KUKA KRL program: EPS_2_26115_SA6999_A_20260219035531.src

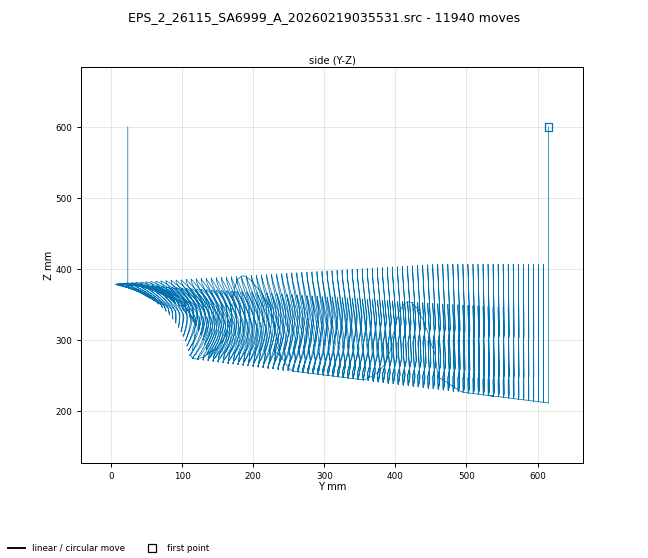
[picture p0: tool path of EPS_2_26115_SA6999_A_20260219035531.src, 11940 of 11942 moves have a stored position in this frame; points joined in program order, loops and branches not executed]
&ACCESS RVP
&REL 4
&COMMENT QRS 19112012
&PARAM EDITMASK = *
DEF PART()
EXT BAS (BAS_COMMAND :IN,REAL :IN )
INT I
BAS (#INITMOV,0 )

;KUKA QRS Post kuka4.cps  Date:22-06-2017 !

File_ID=3054

QRS_PRE_INIT()

;Init var - Until changes are made in qrs_pre_init
Outlet_Square_prg=0
Inlet_1_Square_prg=0
Inlet_2_Square_prg=0
Inlet_3_Square_prg=0
Inlet_4_Square_prg=0
Inlet_5_Square_prg=0

Outlet_1={X 0.000, Y 460.000, Z 306.500, B 0.000, E1 0.000 }
Inlet_1={X 0.000, Y 536.220, Z 246.500, B 0.000, E1 184.000 }
Outlet_1_type=201
Inlet_1_type=201
;QRS#1=Sidecore dimensions
;QRS#2=200-8" PVC SDR 35 Cut Back
;QRS#3=200-8" PVC SDR 35
;QRS#4=
;QRS#5=
;QRS#6=
;QRS#7=
;QRS#8=
;QRS#9=12-08 PSX
;QRS#10=12-08 PSX
;QRS#11=
;QRS#12=
;QRS#13=
;QRS#14=
;QRS#15=
;QRS#16=1220x127x686 2,25'
;QRS#17=EPS Height
;QRS#18=407
;QRS#19=*
;QRS#20= UPDATED VERSION 22-06-2017
;QRS#21=*
Outlet_Square=0100
Inlet_1_Square=0100
Inlet_2_Square=0
Inlet_3_Square=0
Inlet_4_Square=0
Inlet_5_Square=0
Mill_Square=1
Outlet_Square_Prg=214
Inlet_1_Square_prg=204

QRS_INIT()

$ADVANCE=5

; T1
PTP {E1 173.66,E2 173.66}
PTP {X 0,Y 615.427,A -85,B 0,C 180,E1 173.66,E2 173.66,E3 0,E4 0,E5 0,E6 0}
QRS_SPEED_INIT()
LIN {X 0,Y 615.427,Z 600,A -85,B 0,C 180,E1 173.66,E2 173.66,E3 0,E4 0,E5 0,E6 0} C_VEL
LIN {X 0,Y 615.427,Z 221.878,A -85,B 0,C 180,E1 173.66,E2 173.66} C_VEL
LIN {X 0,Y 615.427,Z 213.7,A -85,B 0,C 180,E1 173.66,E2 173.66} C_VEL
LIN {X 0,Y 615.43,Z 211.7,A -85,B 0,C 180,E1 173.474,E2 173.474} C_VEL
LIN {X 0,Y 615.497,Z 211.695,A -85,B 0,C 180,E1 170.801,E2 170.801} C_VEL
LIN {X 0,Y 615.455,Z 211.694,A -85,B 0,C 180,E1 168.138,E2 168.138} C_VEL
LIN {X 0,Y 615.489,Z 211.696,A -85,B 0,C 180,E1 165.451,E2 165.451} C_VEL
LIN {X 0,Y 615.486,Z 211.688,A -85,B 0,C 180,E1 162.729,E2 162.729} C_VEL
LIN {X 0,Y 615.47,Z 211.696,A -85,B 0,C 180,E1 159.966,E2 159.966} C_VEL
LIN {X 0,Y 615.456,Z 211.693,A -85,B 0,C 180,E1 157.663,E2 157.663} C_VEL
LIN {X 0,Y 615.492,Z 211.702,A -85,B 0,C 180,E1 155.008,E2 155.008} C_VEL
LIN {X 0,Y 615.434,Z 211.7,A -85,B 0,C 180,E1 152.082,E2 152.082} C_VEL
LIN {X 0,Y 615.48,Z 211.7,A -85,B 0,C 180,E1 149.839,E2 149.839} C_VEL
LIN {X 0,Y 615.492,Z 211.691,A -85,B 0,C 180,E1 147.543,E2 147.543} C_VEL
LIN {X 0,Y 615.479,Z 211.688,A -85,B 0,C 180,E1 145.184,E2 145.184} C_VEL
LIN {X 0,Y 615.487,Z 211.698,A -85,B 0,C 180,E1 142.757,E2 142.757} C_VEL
LIN {X 0,Y 615.474,Z 211.689,A -85,B 0,C 180,E1 139.914,E2 139.914} C_VEL
LIN {X 0,Y 615.464,Z 211.698,A -85,B 0,C 180,E1 136.956,E2 136.956} C_VEL
LIN {X 0,Y 615.438,Z 211.7,A -85,B 0,C 180,E1 134.926,E2 134.926} C_VEL
LIN {X 0,Y 615.479,Z 211.7,A -85,B 0,C 180,E1 132.079,E2 132.079} C_VEL
LIN {X 0,Y 615.481,Z 211.692,A -85,B 0,C 180,E1 129.752,E2 129.752} C_VEL
LIN {X 0,Y 615.472,Z 211.697,A -85,B 0,C 180,E1 126.934,E2 126.934} C_VEL
LIN {X 0,Y 615.495,Z 211.685,A -85,B 0,C 180,E1 124.022,E2 124.022} C_VEL
LIN {X 0,Y 615.482,Z 211.693,A -85,B 0,C 180,E1 121.687,E2 121.687} C_VEL
LIN {X 0,Y 615.499,Z 213.244,A -85,B 0,C 180,E1 120.16,E2 120.16} C_VEL
LIN {X 0,Y 615.488,Z 215.951,A -85,B 0,C 180,E1 117.916,E2 117.916} C_VEL
LIN {X 0,Y 615.438,Z 218.768,A -85,B 0,C 180,E1 115.558,E2 115.558} C_VEL
LIN {X 0,Y 615.427,Z 221.262,A -85,B 0,C 180,E1 113.56,E2 113.56} C_VEL
LIN {X 0,Y 615.431,Z 224.037,A -85,B 0,C 180,E1 111.435,E2 111.435} C_VEL
LIN {X 0,Y 615.492,Z 227.738,A -85,B 0,C 180,E1 108.647,E2 108.647} C_VEL
LIN {X 0,Y 615.445,Z 231.467,A -85,B 0,C 180,E1 105.907,E2 105.907} C_VEL
LIN {X 0,Y 615.482,Z 235.206,A -85,B 0,C 180,E1 103.202,E2 103.202} C_VEL
LIN {X 0,Y 615.478,Z 238.945,A -85,B 0,C 180,E1 100.528,E2 100.528} C_VEL
LIN {X 0,Y 615.461,Z 242.721,A -85,B 0,C 180,E1 97.877,E2 97.877} C_VEL
LIN {X 0,Y 615.484,Z 243.188,A -85,B 0,C 180,E1 97.546,E2 97.546} C_VEL
LIN {X 0,Y 615.492,Z 257.399,A -85,B 0,C 180,E1 97.217,E2 97.217} C_VEL
LIN {X 0,Y 615.498,Z 269.488,A -85,B 0,C 180,E1 96.809,E2 96.809} C_VEL
LIN {X 0,Y 615.463,Z 280.578,A -85,B 0,C 180,E1 96.311,E2 96.311} C_VEL
LIN {X 0,Y 615.485,Z 291.97,A -85,B 0,C 180,E1 95.653,E2 95.653} C_VEL
LIN {X 0,Y 615.498,Z 302.233,A -85,B 0,C 180,E1 94.914,E2 94.914} C_VEL
LIN {X 0,Y 615.499,Z 311.516,A -85,B 0,C 180,E1 94.093,E2 94.093} C_VEL
LIN {X 0,Y 615.498,Z 320.461,A -85,B 0,C 180,E1 93.11,E2 93.11} C_VEL
LIN {X 0,Y 615.497,Z 327.686,A -85,B 0,C 180,E1 92.128,E2 92.128} C_VEL
LIN {X 0,Y 615.497,Z 334.314,A -85,B 0,C 180,E1 90.982,E2 90.982} C_VEL
LIN {X 0,Y 615.495,Z 338.703,A -85,B 0,C 180,E1 90.001,E2 90.001} C_VEL
LIN {X 0,Y 615.496,Z 341.018,A -85,B 0,C 180,E1 89.347,E2 89.347} C_VEL
LIN {X 0,Y 615.495,Z 342.915,A -85,B 0,C 180,E1 88.692,E2 88.692} C_VEL
LIN {X 0,Y 615.5,Z 344.4,A -85,B 0,C 180,E1 88.038,E2 88.038} C_VEL
LIN {X 0,Y 615.496,Z 346.089,A -85,B 0,C 180,E1 86.728,E2 86.728} C_VEL
LIN {X 0,Y 615.496,Z 346.254,A -85,B 0,C 180,E1 85.417,E2 85.417} C_VEL
LIN {X 0,Y 615.496,Z 344.792,A -85,B 0,C 180,E1 84.103,E2 84.103} C_VEL
LIN {X 0,Y 615.496,Z 343.421,A -85,B 0,C 180,E1 83.418,E2 83.418} C_VEL
LIN {X 0,Y 615.496,Z 340.674,A -85,B 0,C 180,E1 82.456,E2 82.456} C_VEL
LIN {X 0,Y 615.497,Z 336.845,A -85,B 0,C 180,E1 81.465,E2 81.465} C_VEL
LIN {X 0,Y 615.496,Z 331.874,A -85,B 0,C 180,E1 80.471,E2 80.471} C_VEL
LIN {X 0,Y 615.497,Z 325.603,A -85,B 0,C 180,E1 79.474,E2 79.474} C_VEL
LIN {X 0,Y 615.496,Z 317.715,A -85,B 0,C 180,E1 78.474,E2 78.474} C_VEL
LIN {X 0,Y 615.498,Z 309.63,A -85,B 0,C 180,E1 77.639,E2 77.639} C_VEL
LIN {X 0,Y 615.499,Z 299.733,A -85,B 0,C 180,E1 76.8,E2 76.8} C_VEL
LIN {X 0,Y 615.476,Z 289.065,A -85,B 0,C 180,E1 76.073,E2 76.073} C_VEL
LIN {X 0,Y 615.488,Z 277.524,A -85,B 0,C 180,E1 75.452,E2 75.452} C_VEL
LIN {X 0,Y 615.481,Z 265.299,A -85,B 0,C 180,E1 74.944,E2 74.944} C_VEL
LIN {X 0,Y 615.492,Z 252.488,A -85,B 0,C 180,E1 74.563,E2 74.563} C_VEL
LIN {X 0,Y 615.484,Z 243.199,A -85,B 0,C 180,E1 74.372,E2 74.372} C_VEL
LIN {X 0,Y 615.472,Z 239.89,A -85,B 0,C 180,E1 72.044,E2 72.044} C_VEL
LIN {X 0,Y 615.488,Z 235.979,A -85,B 0,C 180,E1 69.27,E2 69.27} C_VEL
LIN {X 0,Y 615.464,Z 232.076,A -85,B 0,C 180,E1 66.444,E2 66.444} C_VEL
LIN {X 0,Y 615.461,Z 229.123,A -85,B 0,C 180,E1 64.284,E2 64.284} C_VEL
LIN {X 0,Y 615.491,Z 225.444,A -85,B 0,C 180,E1 61.55,E2 61.55} C_VEL
LIN {X 0,Y 615.457,Z 222.002,A -85,B 0,C 180,E1 58.919,E2 58.919} C_VEL
LIN {X 0,Y 615.45,Z 218.911,A -85,B 0,C 180,E1 56.472,E2 56.472} C_VEL
LIN {X 0,Y 615.45,Z 215.467,A -85,B 0,C 180,E1 53.574,E2 53.574} C_VEL
LIN {X 0,Y 615.464,Z 212.279,A -85,B 0,C 180,E1 50.941,E2 50.941} C_VEL
LIN {X 0,Y 615.482,Z 211.69,A -85,B 0,C 180,E1 49.912,E2 49.912} C_VEL
LIN {X 0,Y 615.483,Z 211.694,A -85,B 0,C 180,E1 47.648,E2 47.648} C_VEL
LIN {X 0,Y 615.456,Z 211.696,A -85,B 0,C 180,E1 44.93,E2 44.93} C_VEL
LIN {X 0,Y 615.465,Z 211.7,A -85,B 0,C 180,E1 42.08,E2 42.08} C_VEL
LIN {X 0,Y 615.46,Z 211.695,A -85,B 0,C 180,E1 39.753,E2 39.753} C_VEL
LIN {X 0,Y 615.48,Z 211.693,A -85,B 0,C 180,E1 36.938,E2 36.938} C_VEL
LIN {X 0,Y 615.488,Z 211.7,A -85,B 0,C 180,E1 34.022,E2 34.022} C_VEL
LIN {X 0,Y 615.437,Z 211.7,A -85,B 0,C 180,E1 31.689,E2 31.689} C_VEL
LIN {X 0,Y 615.471,Z 211.7,A -85,B 0,C 180,E1 29.407,E2 29.407} C_VEL
LIN {X 0,Y 615.484,Z 211.691,A -85,B 0,C 180,E1 26.445,E2 26.445} C_VEL
LIN {X 0,Y 615.477,Z 211.699,A -85,B 0,C 180,E1 24.009,E2 24.009} C_VEL
LIN {X 0,Y 615.446,Z 211.7,A -85,B 0,C 180,E1 21.434,E2 21.434} C_VEL
LIN {X 0,Y 615.467,Z 211.694,A -85,B 0,C 180,E1 18.603,E2 18.603} C_VEL
LIN {X 0,Y 615.487,Z 211.7,A -85,B 0,C 180,E1 15.905,E2 15.905} C_VEL
LIN {X 0,Y 615.49,Z 211.69,A -85,B 0,C 180,E1 13.201,E2 13.201} C_VEL
LIN {X 0,Y 615.443,Z 211.701,A -85,B 0,C 180,E1 10.528,E2 10.528} C_VEL
LIN {X 0,Y 615.479,Z 211.701,A -85,B 0,C 180,E1 7.876,E2 7.876} C_VEL
LIN {X 0,Y 615.492,Z 211.688,A -85,B 0,C 180,E1 5.241,E2 5.241} C_VEL
LIN {X 0,Y 615.477,Z 211.699,A -85,B 0,C 180,E1 2.618,E2 2.618} C_VEL
LIN {X 0,Y 615.448,Z 211.7,A -85,B 0,C 180,E1 0,E2 0} C_VEL
LIN {X 0,Y 615.48,Z 211.693,A -85,B 0,C 180,E1 -2.618,E2 -2.618} C_VEL
LIN {X 0,Y 615.486,Z 211.698,A -85,B 0,C 180,E1 -5.241,E2 -5.241} C_VEL
LIN {X 0,Y 615.467,Z 211.693,A -85,B 0,C 180,E1 -7.876,E2 -7.876} C_VEL
LIN {X 0,Y 615.478,Z 211.7,A -85,B 0,C 180,E1 -10.527,E2 -10.527} C_VEL
LIN {X 0,Y 615.456,Z 211.699,A -85,B 0,C 180,E1 -13.202,E2 -13.202} C_VEL
LIN {X 0,Y 615.492,Z 211.689,A -85,B 0,C 180,E1 -15.905,E2 -15.905} C_VEL
LIN {X 0,Y 615.489,Z 211.701,A -85,B 0,C 180,E1 -18.646,E2 -18.646} C_VEL
LIN {X 0,Y 615.448,Z 211.7,A -85,B 0,C 180,E1 -20.732,E2 -20.732} C_VEL
LIN {X 0,Y 615.485,Z 211.703,A -85,B 0,C 180,E1 -23.556,E2 -23.556} C_VEL
LIN {X 0,Y 615.476,Z 211.695,A -85,B 0,C 180,E1 -26.445,E2 -26.445} C_VEL
LIN {X 0,Y 615.48,Z 211.699,A -85,B 0,C 180,E1 -28.658,E2 -28.658} C_VEL
LIN {X 0,Y 615.452,Z 211.697,A -85,B 0,C 180,E1 -31.083,E2 -31.083} C_VEL
LIN {X 0,Y 615.456,Z 211.697,A -85,B 0,C 180,E1 -34.024,E2 -34.024} C_VEL
LIN {X 0,Y 615.475,Z 211.697,A -85,B 0,C 180,E1 -36.426,E2 -36.426} C_VEL
LIN {X 0,Y 615.478,Z 211.691,A -85,B 0,C 180,E1 -39.063,E2 -39.063} C_VEL
LIN {X 0,Y 615.497,Z 211.695,A -85,B 0,C 180,E1 -41.473,E2 -41.473} C_VEL
LIN {X 0,Y 615.436,Z 211.7,A -85,B 0,C 180,E1 -44.154,E2 -44.154} C_VEL
LIN {X 0,Y 615.493,Z 211.697,A -85,B 0,C 180,E1 -46.758,E2 -46.758} C_VEL
LIN {X 0,Y 615.483,Z 211.692,A -85,B 0,C 180,E1 -49.395,E2 -49.395} C_VEL
LIN {X 0,Y 615.457,Z 211.698,A -85,B 0,C 180,E1 -51.992,E2 -51.992} C_VEL
LIN {X 0,Y 615.462,Z 211.822,A -85,B 0,C 180,E1 -54.535,E2 -54.535} C_VEL
LIN {X 0,Y 615.471,Z 220.583,A -85,B 0,C 180,E1 -57.154,E2 -57.154} C_VEL
LIN {X 0,Y 615.452,Z 228.516,A -85,B 0,C 180,E1 -59.46,E2 -59.46} C_VEL
LIN {X 0,Y 615.483,Z 237.76,A -85,B 0,C 180,E1 -62.086,E2 -62.086} C_VEL
LIN {X 0,Y 615.488,Z 247.269,A -85,B 0,C 180,E1 -64.721,E2 -64.721} C_VEL
LIN {X 0,Y 615.475,Z 256.241,A -85,B 0,C 180,E1 -67.156,E2 -67.156} C_VEL
LIN {X 0,Y 615.489,Z 264.799,A -85,B 0,C 180,E1 -69.443,E2 -69.443} C_VEL
LIN {X 0,Y 615.49,Z 276.018,A -85,B 0,C 180,E1 -72.388,E2 -72.388} C_VEL
LIN {X 0,Y 615.479,Z 286.546,A -85,B 0,C 180,E1 -75.114,E2 -75.114} C_VEL
LIN {X 0,Y 615.444,Z 295.77,A -85,B 0,C 180,E1 -77.47,E2 -77.47} C_VEL
LIN {X 0,Y 615.499,Z 299.212,A -85,B 0,C 180,E1 -78.349,E2 -78.349} C_VEL
LIN {X 0,Y 615.497,Z 313.861,A -85,B 0,C 180,E1 -78.641,E2 -78.641} C_VEL
LIN {X 0,Y 615.451,Z 327.004,A -85,B 0,C 180,E1 -79.052,E2 -79.052} C_VEL
LIN {X 0,Y 615.438,Z 338.796,A -85,B 0,C 180,E1 -79.556,E2 -79.556} C_VEL
LIN {X 0,Y 615.482,Z 349.407,A -85,B 0,C 180,E1 -80.139,E2 -80.139} C_VEL
LIN {X 0,Y 615.498,Z 360.245,A -85,B 0,C 180,E1 -80.885,E2 -80.885} C_VEL
LIN {X 0,Y 615.497,Z 370.823,A -85,B 0,C 180,E1 -81.795,E2 -81.795} C_VEL
LIN {X 0,Y 615.497,Z 379.974,A -85,B 0,C 180,E1 -82.785,E2 -82.785} C_VEL
LIN {X 0,Y 615.497,Z 387.322,A -85,B 0,C 180,E1 -83.774,E2 -83.774} C_VEL
LIN {X 0,Y 615.498,Z 393.21,A -85,B 0,C 180,E1 -84.76,E2 -84.76} C_VEL
LIN {X 0,Y 615.493,Z 397.856,A -85,B 0,C 180,E1 -85.745,E2 -85.745} C_VEL
LIN {X 0,Y 615.494,Z 401.402,A -85,B 0,C 180,E1 -86.728,E2 -86.728} C_VEL
LIN {X 0,Y 615.497,Z 403.235,A -85,B 0,C 180,E1 -87.383,E2 -87.383} C_VEL
LIN {X 0,Y 615.5,Z 404.609,A -85,B 0,C 180,E1 -88.038,E2 -88.038} C_VEL
LIN {X 0,Y 615.496,Z 406.174,A -85,B 0,C 180,E1 -89.347,E2 -89.347} C_VEL
LIN {X 0,Y 615.494,Z 406.389,A -85,B 0,C 180,E1 -90.001,E2 -90.001} C_VEL
LIN {X 0,Y 615.495,Z 405.579,A -85,B 0,C 180,E1 -91.31,E2 -91.31} C_VEL
LIN {X 0,Y 615.5,Z 404.606,A -85,B 0,C 180,E1 -91.964,E2 -91.964} C_VEL
LIN {X 0,Y 615.497,Z 403.231,A -85,B 0,C 180,E1 -92.619,E2 -92.619} C_VEL
LIN {X 0,Y 615.496,Z 400.346,A -85,B 0,C 180,E1 -93.602,E2 -93.602} C_VEL
LIN {X 0,Y 615.498,Z 396.437,A -85,B 0,C 180,E1 -94.585,E2 -94.585} C_VEL
LIN {X 0,Y 615.499,Z 391.4,A -85,B 0,C 180,E1 -95.571,E2 -95.571} C_VEL
LIN {X 0,Y 615.497,Z 384.869,A -85,B 0,C 180,E1 -96.583,E2 -96.583} C_VEL
LIN {X 0,Y 615.497,Z 377.125,A -85,B 0,C 180,E1 -97.546,E2 -97.546} C_VEL
LIN {X 0,Y 615.498,Z 369.035,A -85,B 0,C 180,E1 -98.372,E2 -98.372} C_VEL
LIN {X 0,Y 615.499,Z 359.155,A -85,B 0,C 180,E1 -99.2,E2 -99.2} C_VEL
LIN {X 0,Y 615.471,Z 347.969,A -85,B 0,C 180,E1 -99.946,E2 -99.946} C_VEL
LIN {X 0,Y 615.437,Z 337.012,A -85,B 0,C 180,E1 -100.529,E2 -100.529} C_VEL
LIN {X 0,Y 615.457,Z 324.782,A -85,B 0,C 180,E1 -101.03,E2 -101.03} C_VEL
LIN {X 0,Y 615.499,Z 312.023,A -85,B 0,C 180,E1 -101.402,E2 -101.402} C_VEL
LIN {X 0,Y 615.498,Z 299.205,A -85,B 0,C 180,E1 -101.653,E2 -101.653} C_VEL
LIN {X 0,Y 615.454,Z 289.085,A -85,B 0,C 180,E1 -104.238,E2 -104.238} C_VEL
LIN {X 0,Y 615.491,Z 278.636,A -85,B 0,C 180,E1 -106.929,E2 -106.929} C_VEL
LIN {X 0,Y 615.482,Z 268.101,A -85,B 0,C 180,E1 -109.686,E2 -109.686} C_VEL
LIN {X 0,Y 615.49,Z 258.087,A -85,B 0,C 180,E1 -112.346,E2 -112.346} C_VEL
LIN {X 0,Y 615.477,Z 248.318,A -85,B 0,C 180,E1 -114.993,E2 -114.993} C_VEL
LIN {X 0,Y 615.492,Z 239.071,A -85,B 0,C 180,E1 -117.546,E2 -117.546} C_VEL
LIN {X 0,Y 615.456,Z 229.83,A -85,B 0,C 180,E1 -120.163,E2 -120.163} C_VEL
LIN {X 0,Y 615.445,Z 221.899,A -85,B 0,C 180,E1 -122.461,E2 -122.461} C_VEL
LIN {X 0,Y 615.491,Z 212.64,A -85,B 0,C 180,E1 -125.215,E2 -125.215} C_VEL
LIN {X 0,Y 615.453,Z 211.7,A -85,B 0,C 180,E1 -125.519,E2 -125.519} C_VEL
LIN {X 0,Y 615.435,Z 211.699,A -85,B 0,C 180,E1 -128.073,E2 -128.073} C_VEL
LIN {X 0,Y 615.495,Z 211.697,A -85,B 0,C 180,E1 -130.607,E2 -130.607} C_VEL
LIN {X 0,Y 615.467,Z 211.691,A -85,B 0,C 180,E1 -133.247,E2 -133.247} C_VEL
LIN {X 0,Y 615.487,Z 211.696,A -85,B 0,C 180,E1 -136.004,E2 -136.004} C_VEL
LIN {X 0,Y 615.489,Z 211.69,A -85,B 0,C 180,E1 -138.906,E2 -138.906} C_VEL
LIN {X 0,Y 615.493,Z 211.701,A -85,B 0,C 180,E1 -141.096,E2 -141.096} C_VEL
LIN {X 0,Y 615.443,Z 211.697,A -85,B 0,C 180,E1 -143.572,E2 -143.572} C_VEL
LIN {X 0,Y 615.492,Z 211.701,A -85,B 0,C 180,E1 -146.466,E2 -146.466} C_VEL
LIN {X 0,Y 615.441,Z 211.697,A -85,B 0,C 180,E1 -149.078,E2 -149.078} C_VEL
LIN {X 0,Y 615.474,Z 211.699,A -85,B 0,C 180,E1 -151.553,E2 -151.553} C_VEL
LIN {X 0,Y 615.482,Z 211.687,A -85,B 0,C 180,E1 -154.434,E2 -154.434} C_VEL
LIN {X 0,Y 615.485,Z 211.701,A -85,B 0,C 180,E1 -157.155,E2 -157.155} C_VEL
LIN {X 0,Y 615.484,Z 211.688,A -85,B 0,C 180,E1 -159.967,E2 -159.967} C_VEL
LIN {X 0,Y 615.461,Z 211.699,A -85,B 0,C 180,E1 -162.729,E2 -162.729} C_VEL
LIN {X 0,Y 615.439,Z 211.699,A -85,B 0,C 180,E1 -164.773,E2 -164.773} C_VEL
LIN {X 0,Y 615.427,Z 211.7,A -85,B 0,C 180,E1 -166.797,E2 -166.797} C_VEL
LIN {X 0,Y 615.489,Z 211.701,A -85,B 0,C 180,E1 -169.473,E2 -169.473} C_VEL
LIN {X 0,Y 615.466,Z 211.691,A -85,B 0,C 180,E1 -172.124,E2 -172.124} C_VEL
LIN {X 0,Y 615.488,Z 211.7,A -85,B 0,C 180,E1 -174.759,E2 -174.759} C_VEL
LIN {X 0,Y 615.487,Z 211.687,A -85,B 0,C 180,E1 -177.382,E2 -177.382} C_VEL
LIN {X 0,Y 615.493,Z 211.697,A -85,B 0,C 180,E1 -180,E2 -180} C_VEL
LIN {X 0,Y 615.449,Z 211.696,A -85,B 0,C 180,E1 -182.618,E2 -182.618} C_VEL
LIN {X 0,Y 615.485,Z 211.696,A -85,B 0,C 180,E1 -185.241,E2 -185.241} C_VEL
LIN {X 0,Y 615.43,Z 211.7,A -85,B 0,C 180,E1 -186.526,E2 -186.526} C_VEL
LIN {X 0,Y 614.797,Z 211.849,A -85,B 0,C 180,E1 -187.072,E2 -187.072} C_VEL
LIN {X 0,Y 612.005,Z 212.247,A -85,B 0,C 180,E1 -187.958,E2 -187.958} C_VEL
LIN {X 0,Y 609.615,Z 212.56,A -85,B 0,C 180,E1 -188.671,E2 -188.671} C_VEL
LIN {X 0,Y 608.56,Z 212.682,A -85,B 0,C 180,E1 -189.22,E2 -189.22} C_VEL
LIN {X 0,Y 608.46,Z 212.691,A -85,B 0,C 180,E1 -189.406,E2 -189.406} C_VEL
LIN {X 0,Y 608.442,Z 212.692,A -85,B 0,C 180,E1 -192,E2 -192} C_VEL
LIN {X 0,Y 608.479,Z 212.689,A -85,B 0,C 180,E1 -194.721,E2 -194.721} C_VEL
LIN {X 0,Y 608.455,Z 212.692,A -85,B 0,C 180,E1 -197.477,E2 -197.477} C_VEL
LIN {X 0,Y 608.448,Z 212.691,A -85,B 0,C 180,E1 -200.275,E2 -200.275} C_VEL
LIN {X 0,Y 608.436,Z 212.692,A -85,B 0,C 180,E1 -202.469,E2 -202.469} C_VEL
LIN {X 0,Y 608.425,Z 212.697,A -85,B 0,C 180,E1 -205.302,E2 -205.302} C_VEL
LIN {X 0,Y 608.432,Z 212.696,A -85,B 0,C 180,E1 -208.268,E2 -208.268} C_VEL
LIN {X 0,Y 608.443,Z 212.695,A -85,B 0,C 180,E1 -210.547,E2 -210.547} C_VEL
LIN {X 0,Y 608.45,Z 212.69,A -85,B 0,C 180,E1 -212.88,E2 -212.88} C_VEL
LIN {X 0,Y 608.447,Z 212.693,A -85,B 0,C 180,E1 -215.278,E2 -215.278} C_VEL
LIN {X 0,Y 608.465,Z 212.691,A -85,B 0,C 180,E1 -217.747,E2 -217.747} C_VEL
LIN {X 0,Y 608.448,Z 212.691,A -85,B 0,C 180,E1 -220.328,E2 -220.328} C_VEL
LIN {X 0,Y 608.435,Z 212.697,A -85,B 0,C 180,E1 -222.962,E2 -222.962} C_VEL
LIN {X 0,Y 608.424,Z 212.694,A -85,B 0,C 180,E1 -225.74,E2 -225.74} C_VEL
LIN {X 0,Y 608.427,Z 212.693,A -85,B 0,C 180,E1 -228.662,E2 -228.662} C_VEL
LIN {X 0,Y 608.424,Z 212.699,A -85,B 0,C 180,E1 -231.408,E2 -231.408} C_VEL
LIN {X 0,Y 608.453,Z 212.691,A -85,B 0,C 180,E1 -233.954,E2 -233.954} C_VEL
LIN {X 0,Y 608.45,Z 212.691,A -85,B 0,C 180,E1 -236.328,E2 -236.328} C_VEL
LIN {X 0,Y 608.42,Z 212.777,A -85,B 0,C 180,E1 -238.737,E2 -238.737} C_VEL
LIN {X 0,Y 608.427,Z 215.467,A -85,B 0,C 180,E1 -240.977,E2 -240.977} C_VEL
LIN {X 0,Y 608.423,Z 219.032,A -85,B 0,C 180,E1 -243.963,E2 -243.963} C_VEL
LIN {X 0,Y 608.395,Z 221.656,A -85,B 0,C 180,E1 -246.151,E2 -246.151} C_VEL
LIN {X 0,Y 608.373,Z 224.447,A -85,B 0,C 180,E1 -248.304,E2 -248.304} C_VEL
LIN {X 0,Y 608.374,Z 227.247,A -85,B 0,C 180,E1 -250.426,E2 -250.426} C_VEL
LIN {X 0,Y 608.412,Z 230.992,A -85,B 0,C 180,E1 -253.214,E2 -253.214} C_VEL
LIN {X 0,Y 608.385,Z 234.831,A -85,B 0,C 180,E1 -256.017,E2 -256.017} C_VEL
LIN {X 0,Y 608.419,Z 238.526,A -85,B 0,C 180,E1 -258.674,E2 -258.674} C_VEL
LIN {X 0,Y 608.409,Z 242.313,A -85,B 0,C 180,E1 -261.362,E2 -261.362} C_VEL
LIN {X 0,Y 608.422,Z 243.754,A -85,B 0,C 180,E1 -262.334,E2 -262.334} C_VEL
LIN {X 0,Y 608.527,Z 256.976,A -85,B 0,C 180,E1 -262.638,E2 -262.638} C_VEL
LIN {X 0,Y 608.527,Z 269.893,A -85,B 0,C 180,E1 -263.076,E2 -263.076} C_VEL
LIN {X 0,Y 608.476,Z 282.377,A -85,B 0,C 180,E1 -263.657,E2 -263.657} C_VEL
LIN {X 0,Y 608.498,Z 294.157,A -85,B 0,C 180,E1 -264.365,E2 -264.365} C_VEL
LIN {X 0,Y 608.476,Z 303.085,A -85,B 0,C 180,E1 -265.03,E2 -265.03} C_VEL
LIN {X 0,Y 608.474,Z 312.286,A -85,B 0,C 180,E1 -265.859,E2 -265.859} C_VEL
LIN {X 0,Y 608.459,Z 321.215,A -85,B 0,C 180,E1 -266.854,E2 -266.854} C_VEL
LIN {X 0,Y 608.454,Z 328.428,A -85,B 0,C 180,E1 -267.848,E2 -267.848} C_VEL
LIN {X 0,Y 608.449,Z 333.311,A -85,B 0,C 180,E1 -268.675,E2 -268.675} C_VEL
LIN {X 0,Y 608.442,Z 338.067,A -85,B 0,C 180,E1 -269.668,E2 -269.668} C_VEL
LIN {X 0,Y 608.439,Z 341.722,A -85,B 0,C 180,E1 -270.661,E2 -270.661} C_VEL
LIN {X 0,Y 608.448,Z 343.613,A -85,B 0,C 180,E1 -271.323,E2 -271.323} C_VEL
LIN {X 0,Y 608.444,Z 345.077,A -85,B 0,C 180,E1 -271.985,E2 -271.985} C_VEL
LIN {X 0,Y 608.422,Z 346.732,A -85,B 0,C 180,E1 -273.31,E2 -273.31} C_VEL
LIN {X 0,Y 608.433,Z 346.989,A -85,B 0,C 180,E1 -273.973,E2 -273.973} C_VEL
LIN {X 0,Y 608.429,Z 346.833,A -85,B 0,C 180,E1 -274.637,E2 -274.637} C_VEL
LIN {X 0,Y 608.433,Z 345.309,A -85,B 0,C 180,E1 -275.966,E2 -275.966} C_VEL
LIN {X 0,Y 608.447,Z 343.956,A -85,B 0,C 180,E1 -276.632,E2 -276.632} C_VEL
LIN {X 0,Y 608.427,Z 341.073,A -85,B 0,C 180,E1 -277.633,E2 -277.633} C_VEL
LIN {X 0,Y 608.431,Z 337.153,A -85,B 0,C 180,E1 -278.635,E2 -278.635} C_VEL
LIN {X 0,Y 608.435,Z 332.078,A -85,B 0,C 180,E1 -279.641,E2 -279.641} C_VEL
LIN {X 0,Y 608.443,Z 325.68,A -85,B 0,C 180,E1 -280.649,E2 -280.649} C_VEL
LIN {X 0,Y 608.474,Z 317.634,A -85,B 0,C 180,E1 -281.66,E2 -281.66} C_VEL
LIN {X 0,Y 608.468,Z 309.411,A -85,B 0,C 180,E1 -282.506,E2 -282.506} C_VEL
LIN {X 0,Y 608.482,Z 299.346,A -85,B 0,C 180,E1 -283.355,E2 -283.355} C_VEL
LIN {X 0,Y 608.479,Z 287.907,A -85,B 0,C 180,E1 -284.121,E2 -284.121} C_VEL
LIN {X 0,Y 608.51,Z 276.663,A -85,B 0,C 180,E1 -284.719,E2 -284.719} C_VEL
LIN {X 0,Y 608.516,Z 264.051,A -85,B 0,C 180,E1 -285.232,E2 -285.232} C_VEL
LIN {X 0,Y 608.552,Z 251.421,A -85,B 0,C 180,E1 -285.596,E2 -285.596} C_VEL
LIN {X 0,Y 608.429,Z 243.67,A -85,B 0,C 180,E1 -285.771,E2 -285.771} C_VEL
LIN {X 0,Y 608.426,Z 239.526,A -85,B 0,C 180,E1 -288.702,E2 -288.702} C_VEL
LIN {X 0,Y 608.416,Z 236.341,A -85,B 0,C 180,E1 -290.982,E2 -290.982} C_VEL
LIN {X 0,Y 608.418,Z 233.383,A -85,B 0,C 180,E1 -293.124,E2 -293.124} C_VEL
LIN {X 0,Y 608.408,Z 229.424,A -85,B 0,C 180,E1 -296.036,E2 -296.036} C_VEL
LIN {X 0,Y 608.426,Z 225.448,A -85,B 0,C 180,E1 -299.021,E2 -299.021} C_VEL
LIN {X 0,Y 608.401,Z 222.454,A -85,B 0,C 180,E1 -301.319,E2 -301.319} C_VEL
LIN {X 0,Y 608.42,Z 219.508,A -85,B 0,C 180,E1 -303.727,E2 -303.727} C_VEL
LIN {X 0,Y 608.436,Z 216.719,A -85,B 0,C 180,E1 -306.091,E2 -306.091} C_VEL
LIN {X 0,Y 608.417,Z 213.704,A -85,B 0,C 180,E1 -308.59,E2 -308.59} C_VEL
LIN {X 0,Y 608.41,Z 212.703,A -85,B 0,C 180,E1 -309.443,E2 -309.443} C_VEL
LIN {X 0,Y 608.465,Z 212.689,A -85,B 0,C 180,E1 -312.059,E2 -312.059} C_VEL
LIN {X 0,Y 608.432,Z 212.695,A -85,B 0,C 180,E1 -314.796,E2 -314.796} C_VEL
LIN {X 0,Y 608.412,Z 212.696,A -85,B 0,C 180,E1 -317.036,E2 -317.036} C_VEL
LIN {X 0,Y 608.445,Z 212.694,A -85,B 0,C 180,E1 -319.696,E2 -319.696} C_VEL
LIN {X 0,Y 608.463,Z 212.692,A -85,B 0,C 180,E1 -322.253,E2 -322.253} C_VEL
LIN {X 0,Y 608.468,Z 212.689,A -85,B 0,C 180,E1 -325.09,E2 -325.09} C_VEL
LIN {X 0,Y 608.448,Z 212.694,A -85,B 0,C 180,E1 -327.904,E2 -327.904} C_VEL
LIN {X 0,Y 608.435,Z 212.693,A -85,B 0,C 180,E1 -330.218,E2 -330.218} C_VEL
LIN {X 0,Y 608.477,Z 212.691,A -85,B 0,C 180,E1 -332.79,E2 -332.79} C_VEL
LIN {X 0,Y 608.453,Z 212.693,A -85,B 0,C 180,E1 -335.429,E2 -335.429} C_VEL
LIN {X 0,Y 608.431,Z 212.693,A -85,B 0,C 180,E1 -338.307,E2 -338.307} C_VEL
LIN {X 0,Y 608.456,Z 212.691,A -85,B 0,C 180,E1 -341.284,E2 -341.284} C_VEL
LIN {X 0,Y 608.457,Z 212.696,A -85,B 0,C 180,E1 -343.906,E2 -343.906} C_VEL
LIN {X 0,Y 608.462,Z 212.69,A -85,B 0,C 180,E1 -346.643,E2 -346.643} C_VEL
LIN {X 0,Y 608.434,Z 212.695,A -85,B 0,C 180,E1 -349.349,E2 -349.349} C_VEL
LIN {X 0,Y 608.466,Z 212.693,A -85,B 0,C 180,E1 -352.033,E2 -352.033} C_VEL
LIN {X 0,Y 608.47,Z 212.688,A -85,B 0,C 180,E1 -354.698,E2 -354.698} C_VEL
LIN {X 0,Y 608.469,Z 212.694,A -85,B 0,C 180,E1 -357.352,E2 -357.352} C_VEL
LIN {X 0,Y 608.441,Z 212.693,A -85,B 0,C 180,E1 -360,E2 -360} C_VEL
LIN {X 0,Y 608.47,Z 212.69,A -85,B 0,C 180,E1 -362.648,E2 -362.648} C_VEL
LIN {X 0,Y 608.464,Z 212.695,A -85,B 0,C 180,E1 -365.302,E2 -365.302} C_VEL
LIN {X 0,Y 608.463,Z 212.689,A -85,B 0,C 180,E1 -367.967,E2 -367.967} C_VEL
LIN {X 0,Y 608.445,Z 212.695,A -85,B 0,C 180,E1 -370.65,E2 -370.65} C_VEL
LIN {X 0,Y 608.443,Z 212.695,A -85,B 0,C 180,E1 -373.357,E2 -373.357} C_VEL
LIN {X 0,Y 608.461,Z 212.69,A -85,B 0,C 180,E1 -376.094,E2 -376.094} C_VEL
LIN {X 0,Y 608.447,Z 212.695,A -85,B 0,C 180,E1 -378.87,E2 -378.87} C_VEL
LIN {X 0,Y 608.441,Z 212.697,A -85,B 0,C 180,E1 -381.693,E2 -381.693} C_VEL
LIN {X 0,Y 608.438,Z 212.693,A -85,B 0,C 180,E1 -384.572,E2 -384.572} C_VEL
LIN {X 0,Y 608.475,Z 212.69,A -85,B 0,C 180,E1 -387.209,E2 -387.209} C_VEL
LIN {X 0,Y 608.475,Z 212.693,A -85,B 0,C 180,E1 -389.975,E2 -389.975} C_VEL
LIN {X 0,Y 608.433,Z 212.694,A -85,B 0,C 180,E1 -392.881,E2 -392.881} C_VEL
LIN {X 0,Y 608.437,Z 212.697,A -85,B 0,C 180,E1 -395.278,E2 -395.278} C_VEL
LIN {X 0,Y 608.466,Z 212.689,A -85,B 0,C 180,E1 -397.747,E2 -397.747} C_VEL
LIN {X 0,Y 608.441,Z 212.695,A -85,B 0,C 180,E1 -400.33,E2 -400.33} C_VEL
LIN {X 0,Y 608.476,Z 212.696,A -85,B 0,C 180,E1 -403.311,E2 -403.311} C_VEL
LIN {X 0,Y 608.448,Z 212.693,A -85,B 0,C 180,E1 -406.13,E2 -406.13} C_VEL
LIN {X 0,Y 608.455,Z 212.691,A -85,B 0,C 180,E1 -408.825,E2 -408.825} C_VEL
LIN {X 0,Y 608.466,Z 212.695,A -85,B 0,C 180,E1 -411.413,E2 -411.413} C_VEL
LIN {X 0,Y 608.426,Z 212.695,A -85,B 0,C 180,E1 -413.957,E2 -413.957} C_VEL
LIN {X 0,Y 608.448,Z 212.82,A -85,B 0,C 180,E1 -414.369,E2 -414.369} C_VEL
LIN {X 0,Y 608.514,Z 221.921,A -85,B 0,C 180,E1 -417.125,E2 -417.125} C_VEL
LIN {X 0,Y 608.499,Z 229.865,A -85,B 0,C 180,E1 -419.458,E2 -419.458} C_VEL
LIN {X 0,Y 608.495,Z 239.132,A -85,B 0,C 180,E1 -422.112,E2 -422.112} C_VEL
LIN {X 0,Y 608.479,Z 248.399,A -85,B 0,C 180,E1 -424.702,E2 -424.702} C_VEL
LIN {X 0,Y 608.476,Z 258.99,A -85,B 0,C 180,E1 -427.596,E2 -427.596} C_VEL
LIN {X 0,Y 608.457,Z 269.581,A -85,B 0,C 180,E1 -430.431,E2 -430.431} C_VEL
LIN {X 0,Y 608.449,Z 280.173,A -85,B 0,C 180,E1 -433.217,E2 -433.217} C_VEL
LIN {X 0,Y 608.435,Z 290.896,A -85,B 0,C 180,E1 -435.997,E2 -435.997} C_VEL
LIN {X 0,Y 608.437,Z 299.576,A -85,B 0,C 180,E1 -438.223,E2 -438.223} C_VEL
LIN {X 0,Y 608.549,Z 313.14,A -85,B 0,C 180,E1 -438.489,E2 -438.489} C_VEL
LIN {X 0,Y 608.485,Z 325.548,A -85,B 0,C 180,E1 -438.866,E2 -438.866} C_VEL
LIN {X 0,Y 608.444,Z 337.194,A -85,B 0,C 180,E1 -439.351,E2 -439.351} C_VEL
LIN {X 0,Y 608.471,Z 349.596,A -85,B 0,C 180,E1 -440.024,E2 -440.024} C_VEL
LIN {X 0,Y 608.483,Z 360.487,A -85,B 0,C 180,E1 -440.779,E2 -440.779} C_VEL
LIN {X 0,Y 608.474,Z 371.123,A -85,B 0,C 180,E1 -441.7,E2 -441.7} C_VEL
LIN {X 0,Y 608.47,Z 378.969,A -85,B 0,C 180,E1 -442.535,E2 -442.535} C_VEL
LIN {X 0,Y 608.46,Z 386.29,A -85,B 0,C 180,E1 -443.485,E2 -443.485} C_VEL
LIN {X 0,Y 608.45,Z 391.871,A -85,B 0,C 180,E1 -444.367,E2 -444.367} C_VEL
LIN {X 0,Y 608.432,Z 396.954,A -85,B 0,C 180,E1 -445.363,E2 -445.363} C_VEL
LIN {X 0,Y 608.449,Z 400.899,A -85,B 0,C 180,E1 -446.359,E2 -446.359} C_VEL
LIN {X 0,Y 608.425,Z 403.812,A -85,B 0,C 180,E1 -447.353,E2 -447.353} C_VEL
LIN {X 0,Y 608.444,Z 405.203,A -85,B 0,C 180,E1 -448.015,E2 -448.015} C_VEL
LIN {X 0,Y 608.438,Z 406.784,A -85,B 0,C 180,E1 -449.339,E2 -449.339} C_VEL
LIN {X 0,Y 608.434,Z 407,A -85,B 0,C 180,E1 -450.001,E2 -450.001} C_VEL
LIN {X 0,Y 608.448,Z 406.183,A -85,B 0,C 180,E1 -451.325,E2 -451.325} C_VEL
LIN {X 0,Y 608.445,Z 405.2,A -85,B 0,C 180,E1 -451.987,E2 -451.987} C_VEL
LIN {X 0,Y 608.425,Z 403.807,A -85,B 0,C 180,E1 -452.649,E2 -452.649} C_VEL
LIN {X 0,Y 608.449,Z 400.893,A -85,B 0,C 180,E1 -453.643,E2 -453.643} C_VEL
LIN {X 0,Y 608.432,Z 396.946,A -85,B 0,C 180,E1 -454.639,E2 -454.639} C_VEL
LIN {X 0,Y 608.438,Z 390.871,A -85,B 0,C 180,E1 -455.802,E2 -455.802} C_VEL
LIN {X 0,Y 608.463,Z 384.228,A -85,B 0,C 180,E1 -456.8,E2 -456.8} C_VEL
LIN {X 0,Y 608.456,Z 375.981,A -85,B 0,C 180,E1 -457.801,E2 -457.801} C_VEL
LIN {X 0,Y 608.472,Z 367.525,A -85,B 0,C 180,E1 -458.637,E2 -458.637} C_VEL
LIN {X 0,Y 608.48,Z 357.078,A -85,B 0,C 180,E1 -459.474,E2 -459.474} C_VEL
LIN {X 0,Y 608.482,Z 346.74,A -85,B 0,C 180,E1 -460.146,E2 -460.146} C_VEL
LIN {X 0,Y 608.463,Z 335.863,A -85,B 0,C 180,E1 -460.713,E2 -460.713} C_VEL
LIN {X 0,Y 608.492,Z 324.079,A -85,B 0,C 180,E1 -461.187,E2 -461.187} C_VEL
LIN {X 0,Y 608.551,Z 311.227,A -85,B 0,C 180,E1 -461.555,E2 -461.555} C_VEL
LIN {X 0,Y 608.439,Z 299.527,A -85,B 0,C 180,E1 -461.79,E2 -461.79} C_VEL
LIN {X 0,Y 608.405,Z 289.432,A -85,B 0,C 180,E1 -464.381,E2 -464.381} C_VEL
LIN {X 0,Y 608.451,Z 280.165,A -85,B 0,C 180,E1 -466.785,E2 -466.785} C_VEL
LIN {X 0,Y 608.458,Z 269.574,A -85,B 0,C 180,E1 -469.571,E2 -469.571} C_VEL
LIN {X 0,Y 608.465,Z 258.722,A -85,B 0,C 180,E1 -472.477,E2 -472.477} C_VEL
LIN {X 0,Y 608.479,Z 248.391,A -85,B 0,C 180,E1 -475.301,E2 -475.301} C_VEL
LIN {X 0,Y 608.496,Z 239.124,A -85,B 0,C 180,E1 -477.89,E2 -477.89} C_VEL
LIN {X 0,Y 608.481,Z 229.857,A -85,B 0,C 180,E1 -480.545,E2 -480.545} C_VEL
LIN {X 0,Y 608.528,Z 220.59,A -85,B 0,C 180,E1 -483.271,E2 -483.271} C_VEL
LIN {X 0,Y 608.426,Z 212.697,A -85,B 0,C 180,E1 -485.673,E2 -485.673} C_VEL
LIN {X 0,Y 608.434,Z 212.694,A -85,B 0,C 180,E1 -488.236,E2 -488.236} C_VEL
LIN {X 0,Y 608.44,Z 212.691,A -85,B 0,C 180,E1 -491.179,E2 -491.179} C_VEL
LIN {X 0,Y 608.469,Z 212.694,A -85,B 0,C 180,E1 -493.87,E2 -493.87} C_VEL
LIN {X 0,Y 608.483,Z 212.686,A -85,B 0,C 180,E1 -496.691,E2 -496.691} C_VEL
LIN {X 0,Y 608.459,Z 212.692,A -85,B 0,C 180,E1 -499.697,E2 -499.697} C_VEL
LIN {X 0,Y 608.481,Z 212.694,A -85,B 0,C 180,E1 -502.841,E2 -502.841} C_VEL
LIN {X 0,Y 608.426,Z 212.693,A -85,B 0,C 180,E1 -505.528,E2 -505.528} C_VEL
LIN {X 0,Y 608.439,Z 212.695,A -85,B 0,C 180,E1 -507.904,E2 -507.904} C_VEL
LIN {X 0,Y 608.481,Z 212.691,A -85,B 0,C 180,E1 -510.221,E2 -510.221} C_VEL
LIN {X 0,Y 608.438,Z 212.695,A -85,B 0,C 180,E1 -513.225,E2 -513.225} C_VEL
LIN {X 0,Y 608.478,Z 212.688,A -85,B 0,C 180,E1 -515.849,E2 -515.849} C_VEL
LIN {X 0,Y 608.468,Z 212.689,A -85,B 0,C 180,E1 -518.308,E2 -518.308} C_VEL
LIN {X 0,Y 608.447,Z 212.692,A -85,B 0,C 180,E1 -521.13,E2 -521.13} C_VEL
LIN {X 0,Y 608.454,Z 212.694,A -85,B 0,C 180,E1 -523.906,E2 -523.906} C_VEL
LIN {X 0,Y 608.42,Z 212.694,A -85,B 0,C 180,E1 -526.643,E2 -526.643} C_VEL
LIN {X 0,Y 608.454,Z 212.695,A -85,B 0,C 180,E1 -529.35,E2 -529.35} C_VEL
LIN {X 0,Y 608.437,Z 212.692,A -85,B 0,C 180,E1 -532.033,E2 -532.033} C_VEL
LIN {X 0,Y 608.467,Z 212.694,A -85,B 0,C 180,E1 -534.698,E2 -534.698} C_VEL
LIN {X 0,Y 608.478,Z 212.686,A -85,B 0,C 180,E1 -537.352,E2 -537.352} C_VEL
LIN {X 0,Y 608.484,Z 212.692,A -85,B 0,C 180,E1 -540,E2 -540} C_VEL
LIN {X 0,Y 608.445,Z 212.691,A -85,B 0,C 180,E1 -542.648,E2 -542.648} C_VEL
LIN {X 0,Y 608.461,Z 212.694,A -85,B 0,C 180,E1 -545.302,E2 -545.302} C_VEL
LIN {X 0,Y 608.406,Z 212.695,A -85,B 0,C 180,E1 -547.968,E2 -547.968} C_VEL
LIN {X 0,Y 608.46,Z 212.691,A -85,B 0,C 180,E1 -549.406,E2 -549.406} C_VEL
LIN {X 0,Y 607.755,Z 212.778,A -85,B 0,C 180,E1 -549.959,E2 -549.959} C_VEL
LIN {X 0,Y 604.894,Z 213.141,A -85,B 0,C 180,E1 -550.856,E2 -550.856} C_VEL
LIN {X 0,Y 602.504,Z 213.436,A -85,B 0,C 180,E1 -551.577,E2 -551.577} C_VEL
LIN {X 0,Y 601.484,Z 213.56,A -85,B 0,C 180,E1 -552.134,E2 -552.134} C_VEL
LIN {X 0,Y 601.403,Z 213.57,A -85,B 0,C 180,E1 -552.322,E2 -552.322} C_VEL
LIN {X 0,Y 601.434,Z 213.565,A -85,B 0,C 180,E1 -554.897,E2 -554.897} C_VEL
LIN {X 0,Y 601.419,Z 213.566,A -85,B 0,C 180,E1 -556.986,E2 -556.986} C_VEL
LIN {X 0,Y 601.401,Z 213.574,A -85,B 0,C 180,E1 -559.81,E2 -559.81} C_VEL
LIN {X 0,Y 601.408,Z 213.569,A -85,B 0,C 180,E1 -562.683,E2 -562.683} C_VEL
LIN {X 0,Y 601.386,Z 213.577,A -85,B 0,C 180,E1 -564.88,E2 -564.88} C_VEL
LIN {X 0,Y 601.377,Z 213.572,A -85,B 0,C 180,E1 -567.354,E2 -567.354} C_VEL
LIN {X 0,Y 601.384,Z 213.57,A -85,B 0,C 180,E1 -569.395,E2 -569.395} C_VEL
LIN {X 0,Y 601.401,Z 213.571,A -85,B 0,C 180,E1 -571.727,E2 -571.727} C_VEL
LIN {X 0,Y 601.426,Z 213.569,A -85,B 0,C 180,E1 -574.119,E2 -574.119} C_VEL
LIN {X 0,Y 601.404,Z 213.568,A -85,B 0,C 180,E1 -576.583,E2 -576.583} C_VEL
LIN {X 0,Y 601.41,Z 213.575,A -85,B 0,C 180,E1 -579.127,E2 -579.127} C_VEL
LIN {X 0,Y 601.417,Z 213.566,A -85,B 0,C 180,E1 -581.766,E2 -581.766} C_VEL
LIN {X 0,Y 601.405,Z 213.576,A -85,B 0,C 180,E1 -584.532,E2 -584.532} C_VEL
LIN {X 0,Y 601.357,Z 213.574,A -85,B 0,C 180,E1 -587.324,E2 -587.324} C_VEL
LIN {X 0,Y 601.404,Z 213.573,A -85,B 0,C 180,E1 -590.003,E2 -590.003} C_VEL
LIN {X 0,Y 601.436,Z 213.564,A -85,B 0,C 180,E1 -592.618,E2 -592.618} C_VEL
LIN {X 0,Y 601.418,Z 213.573,A -85,B 0,C 180,E1 -595.067,E2 -595.067} C_VEL
LIN {X 0,Y 601.427,Z 213.566,A -85,B 0,C 180,E1 -597.483,E2 -597.483} C_VEL
LIN {X 0,Y 601.345,Z 213.809,A -85,B 0,C 180,E1 -599.053,E2 -599.053} C_VEL
LIN {X 0,Y 601.358,Z 216.577,A -85,B 0,C 180,E1 -601.368,E2 -601.368} C_VEL
LIN {X 0,Y 601.344,Z 219.852,A -85,B 0,C 180,E1 -604.147,E2 -604.147} C_VEL
LIN {X 0,Y 601.304,Z 222.744,A -85,B 0,C 180,E1 -606.584,E2 -606.584} C_VEL
LIN {X 0,Y 601.343,Z 226.385,A -85,B 0,C 180,E1 -609.474,E2 -609.474} C_VEL
LIN {X 0,Y 601.311,Z 229.19,A -85,B 0,C 180,E1 -611.604,E2 -611.604} C_VEL
LIN {X 0,Y 601.33,Z 232.002,A -85,B 0,C 180,E1 -613.709,E2 -613.709} C_VEL
LIN {X 0,Y 601.311,Z 235.765,A -85,B 0,C 180,E1 -616.481,E2 -616.481} C_VEL
LIN {X 0,Y 601.333,Z 239.541,A -85,B 0,C 180,E1 -619.221,E2 -619.221} C_VEL
LIN {X 0,Y 601.318,Z 243.568,A -85,B 0,C 180,E1 -622.106,E2 -622.106} C_VEL
LIN {X 0,Y 601.308,Z 243.687,A -85,B 0,C 180,E1 -622.19,E2 -622.19} C_VEL
LIN {X 0,Y 601.606,Z 247.938,A -85,B 0,C 180,E1 -622.278,E2 -622.278} C_VEL
LIN {X 0,Y 601.568,Z 260.67,A -85,B 0,C 180,E1 -622.616,E2 -622.616} C_VEL
LIN {X 0,Y 601.551,Z 273.95,A -85,B 0,C 180,E1 -623.121,E2 -623.121} C_VEL
LIN {X 0,Y 601.48,Z 285.059,A -85,B 0,C 180,E1 -623.68,E2 -623.68} C_VEL
LIN {X 0,Y 601.468,Z 296.038,A -85,B 0,C 180,E1 -624.383,E2 -624.383} C_VEL
LIN {X 0,Y 601.44,Z 305.612,A -85,B 0,C 180,E1 -625.139,E2 -625.139} C_VEL
LIN {X 0,Y 601.401,Z 314.362,A -85,B 0,C 180,E1 -625.978,E2 -625.978} C_VEL
LIN {X 0,Y 601.384,Z 322.91,A -85,B 0,C 180,E1 -626.985,E2 -626.985} C_VEL
LIN {X 0,Y 601.355,Z 329.761,A -85,B 0,C 180,E1 -627.99,E2 -627.99} C_VEL
LIN {X 0,Y 601.382,Z 335.259,A -85,B 0,C 180,E1 -628.995,E2 -628.995} C_VEL
LIN {X 0,Y 601.357,Z 339.584,A -85,B 0,C 180,E1 -629.999,E2 -629.999} C_VEL
LIN {X 0,Y 601.341,Z 341.873,A -85,B 0,C 180,E1 -630.669,E2 -630.669} C_VEL
LIN {X 0,Y 601.348,Z 343.74,A -85,B 0,C 180,E1 -631.338,E2 -631.338} C_VEL
LIN {X 0,Y 601.343,Z 345.156,A -85,B 0,C 180,E1 -632.008,E2 -632.008} C_VEL
LIN {X 0,Y 601.338,Z 346.766,A -85,B 0,C 180,E1 -633.349,E2 -633.349} C_VEL
LIN {X 0,Y 601.342,Z 346.999,A -85,B 0,C 180,E1 -634.02,E2 -634.02} C_VEL
LIN {X 0,Y 601.336,Z 346.208,A -85,B 0,C 180,E1 -635.364,E2 -635.364} C_VEL
LIN {X 0,Y 601.362,Z 344.103,A -85,B 0,C 180,E1 -636.594,E2 -636.594} C_VEL
LIN {X 0,Y 601.339,Z 340.92,A -85,B 0,C 180,E1 -637.723,E2 -637.723} C_VEL
LIN {X 0,Y 601.35,Z 336.949,A -85,B 0,C 180,E1 -638.738,E2 -638.738} C_VEL
LIN {X 0,Y 601.361,Z 330.812,A -85,B 0,C 180,E1 -639.925,E2 -639.925} C_VEL
LIN {X 0,Y 601.386,Z 323.751,A -85,B 0,C 180,E1 -640.991,E2 -640.991} C_VEL
LIN {X 0,Y 601.43,Z 315.698,A -85,B 0,C 180,E1 -641.97,E2 -641.97} C_VEL
LIN {X 0,Y 601.426,Z 307.032,A -85,B 0,C 180,E1 -642.827,E2 -642.827} C_VEL
LIN {X 0,Y 601.476,Z 296.842,A -85,B 0,C 180,E1 -643.648,E2 -643.648} C_VEL
LIN {X 0,Y 601.503,Z 285.652,A -85,B 0,C 180,E1 -644.375,E2 -644.375} C_VEL
LIN {X 0,Y 601.528,Z 273.702,A -85,B 0,C 180,E1 -644.98,E2 -644.98} C_VEL
LIN {X 0,Y 601.54,Z 261.232,A -85,B 0,C 180,E1 -645.457,E2 -645.457} C_VEL
LIN {X 0,Y 601.599,Z 248.366,A -85,B 0,C 180,E1 -645.802,E2 -645.802} C_VEL
LIN {X 0,Y 601.328,Z 243.711,A -85,B 0,C 180,E1 -645.897,E2 -645.897} C_VEL
LIN {X 0,Y 601.342,Z 239.64,A -85,B 0,C 180,E1 -648.796,E2 -648.796} C_VEL
LIN {X 0,Y 601.311,Z 236.268,A -85,B 0,C 180,E1 -651.242,E2 -651.242} C_VEL
LIN {X 0,Y 601.332,Z 233.309,A -85,B 0,C 180,E1 -653.413,E2 -653.413} C_VEL
LIN {X 0,Y 601.312,Z 230.04,A -85,B 0,C 180,E1 -655.847,E2 -655.847} C_VEL
LIN {X 0,Y 601.343,Z 226.366,A -85,B 0,C 180,E1 -658.63,E2 -658.63} C_VEL
LIN {X 0,Y 601.334,Z 222.781,A -85,B 0,C 180,E1 -661.441,E2 -661.441} C_VEL
LIN {X 0,Y 601.353,Z 219.686,A -85,B 0,C 180,E1 -664.122,E2 -664.122} C_VEL
LIN {X 0,Y 601.333,Z 216.757,A -85,B 0,C 180,E1 -666.586,E2 -666.586} C_VEL
LIN {X 0,Y 601.37,Z 213.729,A -85,B 0,C 180,E1 -669.128,E2 -669.128} C_VEL
LIN {X 0,Y 601.424,Z 213.566,A -85,B 0,C 180,E1 -671.764,E2 -671.764} C_VEL
LIN {X 0,Y 601.419,Z 213.572,A -85,B 0,C 180,E1 -674.534,E2 -674.534} C_VEL
LIN {X 0,Y 601.405,Z 213.573,A -85,B 0,C 180,E1 -677.408,E2 -677.408} C_VEL
LIN {X 0,Y 601.406,Z 213.57,A -85,B 0,C 180,E1 -680.466,E2 -680.466} C_VEL
LIN {X 0,Y 601.43,Z 213.573,A -85,B 0,C 180,E1 -682.617,E2 -682.617} C_VEL
LIN {X 0,Y 601.426,Z 213.566,A -85,B 0,C 180,E1 -685.068,E2 -685.068} C_VEL
LIN {X 0,Y 601.431,Z 213.572,A -85,B 0,C 180,E1 -687.484,E2 -687.484} C_VEL
LIN {X 0,Y 601.4,Z 213.573,A -85,B 0,C 180,E1 -690.606,E2 -690.606} C_VEL
LIN {X 0,Y 601.449,Z 213.565,A -85,B 0,C 180,E1 -692.889,E2 -692.889} C_VEL
LIN {X 0,Y 601.451,Z 213.569,A -85,B 0,C 180,E1 -695.859,E2 -695.859} C_VEL
LIN {X 0,Y 601.384,Z 213.574,A -85,B 0,C 180,E1 -698.76,E2 -698.76} C_VEL
LIN {X 0,Y 601.388,Z 213.571,A -85,B 0,C 180,E1 -701.607,E2 -701.607} C_VEL
LIN {X 0,Y 601.433,Z 213.568,A -85,B 0,C 180,E1 -703.713,E2 -703.713} C_VEL
LIN {X 0,Y 601.413,Z 213.568,A -85,B 0,C 180,E1 -706.484,E2 -706.484} C_VEL
LIN {X 0,Y 601.404,Z 213.572,A -85,B 0,C 180,E1 -709.224,E2 -709.224} C_VEL
LIN {X 0,Y 601.427,Z 213.569,A -85,B 0,C 180,E1 -711.939,E2 -711.939} C_VEL
LIN {X 0,Y 601.434,Z 213.565,A -85,B 0,C 180,E1 -714.636,E2 -714.636} C_VEL
LIN {X 0,Y 601.434,Z 213.57,A -85,B 0,C 180,E1 -717.321,E2 -717.321} C_VEL
LIN {X 0,Y 601.412,Z 213.569,A -85,B 0,C 180,E1 -720,E2 -720} C_VEL
LIN {X 0,Y 601.434,Z 213.566,A -85,B 0,C 180,E1 -722.679,E2 -722.679} C_VEL
LIN {X 0,Y 601.426,Z 213.573,A -85,B 0,C 180,E1 -725.364,E2 -725.364} C_VEL
LIN {X 0,Y 601.428,Z 213.566,A -85,B 0,C 180,E1 -728.061,E2 -728.061} C_VEL
LIN {X 0,Y 601.39,Z 213.571,A -85,B 0,C 180,E1 -731.002,E2 -731.002} C_VEL
LIN {X 0,Y 601.401,Z 213.574,A -85,B 0,C 180,E1 -733.516,E2 -733.516} C_VEL
LIN {X 0,Y 601.435,Z 213.565,A -85,B 0,C 180,E1 -736.287,E2 -736.287} C_VEL
LIN {X 0,Y 601.407,Z 213.569,A -85,B 0,C 180,E1 -739.099,E2 -739.099} C_VEL
LIN {X 0,Y 601.38,Z 213.572,A -85,B 0,C 180,E1 -741.24,E2 -741.24} C_VEL
LIN {X 0,Y 601.445,Z 213.564,A -85,B 0,C 180,E1 -744.141,E2 -744.141} C_VEL
LIN {X 0,Y 601.447,Z 213.567,A -85,B 0,C 180,E1 -747.111,E2 -747.111} C_VEL
LIN {X 0,Y 601.42,Z 213.567,A -85,B 0,C 180,E1 -749.393,E2 -749.393} C_VEL
LIN {X 0,Y 601.385,Z 213.578,A -85,B 0,C 180,E1 -751.728,E2 -751.728} C_VEL
LIN {X 0,Y 601.415,Z 213.568,A -85,B 0,C 180,E1 -754.119,E2 -754.119} C_VEL
LIN {X 0,Y 601.399,Z 213.575,A -85,B 0,C 180,E1 -756.583,E2 -756.583} C_VEL
LIN {X 0,Y 601.435,Z 213.566,A -85,B 0,C 180,E1 -759.537,E2 -759.537} C_VEL
LIN {X 0,Y 601.408,Z 213.574,A -85,B 0,C 180,E1 -761.767,E2 -761.767} C_VEL
LIN {X 0,Y 601.389,Z 213.572,A -85,B 0,C 180,E1 -764.533,E2 -764.533} C_VEL
LIN {X 0,Y 601.406,Z 213.569,A -85,B 0,C 180,E1 -767.41,E2 -767.41} C_VEL
LIN {X 0,Y 601.41,Z 213.574,A -85,B 0,C 180,E1 -770.006,E2 -770.006} C_VEL
LIN {X 0,Y 601.428,Z 213.567,A -85,B 0,C 180,E1 -772.619,E2 -772.619} C_VEL
LIN {X 0,Y 601.402,Z 213.692,A -85,B 0,C 180,E1 -774.159,E2 -774.159} C_VEL
LIN {X 0,Y 601.541,Z 219.274,A -85,B 0,C 180,E1 -775.89,E2 -775.89} C_VEL
LIN {X 0,Y 601.561,Z 228.025,A -85,B 0,C 180,E1 -778.524,E2 -778.524} C_VEL
LIN {X 0,Y 601.478,Z 237.808,A -85,B 0,C 180,E1 -781.377,E2 -781.377} C_VEL
LIN {X 0,Y 601.477,Z 247.454,A -85,B 0,C 180,E1 -784.121,E2 -784.121} C_VEL
LIN {X 0,Y 601.465,Z 256.342,A -85,B 0,C 180,E1 -786.593,E2 -786.593} C_VEL
LIN {X 0,Y 601.43,Z 266.934,A -85,B 0,C 180,E1 -789.479,E2 -789.479} C_VEL
LIN {X 0,Y 601.4,Z 277.525,A -85,B 0,C 180,E1 -792.313,E2 -792.313} C_VEL
LIN {X 0,Y 601.365,Z 288.116,A -85,B 0,C 180,E1 -795.103,E2 -795.103} C_VEL
LIN {X 0,Y 601.338,Z 297.383,A -85,B 0,C 180,E1 -797.514,E2 -797.514} C_VEL
LIN {X 0,Y 601.372,Z 299.534,A -85,B 0,C 180,E1 -798.072,E2 -798.072} C_VEL
LIN {X 0,Y 601.592,Z 313.14,A -85,B 0,C 180,E1 -798.354,E2 -798.354} C_VEL
LIN {X 0,Y 601.509,Z 326.352,A -85,B 0,C 180,E1 -798.766,E2 -798.766} C_VEL
LIN {X 0,Y 601.468,Z 338.944,A -85,B 0,C 180,E1 -799.311,E2 -799.311} C_VEL
LIN {X 0,Y 601.461,Z 349.597,A -85,B 0,C 180,E1 -799.907,E2 -799.907} C_VEL
LIN {X 0,Y 601.449,Z 360.488,A -85,B 0,C 180,E1 -800.67,E2 -800.67} C_VEL
LIN {X 0,Y 601.429,Z 371.123,A -85,B 0,C 180,E1 -801.602,E2 -801.602} C_VEL
LIN {X 0,Y 601.417,Z 378.969,A -85,B 0,C 180,E1 -802.447,E2 -802.447} C_VEL
LIN {X 0,Y 601.369,Z 386.23,A -85,B 0,C 180,E1 -803.399,E2 -803.399} C_VEL
LIN {X 0,Y 601.372,Z 391.872,A -85,B 0,C 180,E1 -804.3,E2 -804.3} C_VEL
LIN {X 0,Y 601.336,Z 396.954,A -85,B 0,C 180,E1 -805.308,E2 -805.308} C_VEL
LIN {X 0,Y 601.368,Z 400.899,A -85,B 0,C 180,E1 -806.316,E2 -806.316} C_VEL
LIN {X 0,Y 601.325,Z 403.812,A -85,B 0,C 180,E1 -807.321,E2 -807.321} C_VEL
LIN {X 0,Y 601.343,Z 405.203,A -85,B 0,C 180,E1 -807.992,E2 -807.992} C_VEL
LIN {X 0,Y 601.339,Z 406.784,A -85,B 0,C 180,E1 -809.331,E2 -809.331} C_VEL
LIN {X 0,Y 601.335,Z 407,A -85,B 0,C 180,E1 -810.001,E2 -810.001} C_VEL
LIN {X 0,Y 601.347,Z 406.183,A -85,B 0,C 180,E1 -811.34,E2 -811.34} C_VEL
LIN {X 0,Y 601.343,Z 405.2,A -85,B 0,C 180,E1 -812.01,E2 -812.01} C_VEL
LIN {X 0,Y 601.325,Z 403.807,A -85,B 0,C 180,E1 -812.681,E2 -812.681} C_VEL
LIN {X 0,Y 601.368,Z 400.893,A -85,B 0,C 180,E1 -813.686,E2 -813.686} C_VEL
LIN {X 0,Y 601.336,Z 396.946,A -85,B 0,C 180,E1 -814.694,E2 -814.694} C_VEL
LIN {X 0,Y 601.373,Z 390.871,A -85,B 0,C 180,E1 -815.87,E2 -815.87} C_VEL
LIN {X 0,Y 601.382,Z 384.228,A -85,B 0,C 180,E1 -816.881,E2 -816.881} C_VEL
LIN {X 0,Y 601.401,Z 375.981,A -85,B 0,C 180,E1 -817.893,E2 -817.893} C_VEL
LIN {X 0,Y 601.436,Z 367.526,A -85,B 0,C 180,E1 -818.739,E2 -818.739} C_VEL
LIN {X 0,Y 601.447,Z 357.078,A -85,B 0,C 180,E1 -819.586,E2 -819.586} C_VEL
LIN {X 0,Y 601.473,Z 346.74,A -85,B 0,C 180,E1 -820.265,E2 -820.265} C_VEL
LIN {X 0,Y 601.482,Z 335.241,A -85,B 0,C 180,E1 -820.868,E2 -820.868} C_VEL
LIN {X 0,Y 601.528,Z 322.313,A -85,B 0,C 180,E1 -821.376,E2 -821.376} C_VEL
LIN {X 0,Y 601.597,Z 309.399,A -85,B 0,C 180,E1 -821.733,E2 -821.733} C_VEL
LIN {X 0,Y 601.373,Z 299.527,A -85,B 0,C 180,E1 -821.93,E2 -821.93} C_VEL
LIN {X 0,Y 601.37,Z 289.432,A -85,B 0,C 180,E1 -824.553,E2 -824.553} C_VEL
LIN {X 0,Y 601.396,Z 278.841,A -85,B 0,C 180,E1 -827.338,E2 -827.338} C_VEL
LIN {X 0,Y 601.421,Z 268.25,A -85,B 0,C 180,E1 -830.166,E2 -830.166} C_VEL
LIN {X 0,Y 601.436,Z 258.983,A -85,B 0,C 180,E1 -832.683,E2 -832.683} C_VEL
LIN {X 0,Y 601.463,Z 249.715,A -85,B 0,C 180,E1 -835.246,E2 -835.246} C_VEL
LIN {X 0,Y 601.504,Z 240.448,A -85,B 0,C 180,E1 -837.864,E2 -837.864} C_VEL
LIN {X 0,Y 601.507,Z 231.181,A -85,B 0,C 180,E1 -840.548,E2 -840.548} C_VEL
LIN {X 0,Y 601.585,Z 221.914,A -85,B 0,C 180,E1 -843.305,E2 -843.305} C_VEL
LIN {X 0,Y 601.585,Z 215.919,A -85,B 0,C 180,E1 -845.137,E2 -845.137} C_VEL
LIN {X 0,Y 601.388,Z 213.574,A -85,B 0,C 180,E1 -845.933,E2 -845.933} C_VEL
LIN {X 0,Y 601.4,Z 213.574,A -85,B 0,C 180,E1 -848.467,E2 -848.467} C_VEL
LIN {X 0,Y 601.405,Z 213.57,A -85,B 0,C 180,E1 -850.876,E2 -850.876} C_VEL
LIN {X 0,Y 601.412,Z 213.569,A -85,B 0,C 180,E1 -853.589,E2 -853.589} C_VEL
LIN {X 0,Y 601.436,Z 213.564,A -85,B 0,C 180,E1 -856.428,E2 -856.428} C_VEL
LIN {X 0,Y 601.415,Z 213.571,A -85,B 0,C 180,E1 -859.125,E2 -859.125} C_VEL
LIN {X 0,Y 601.4,Z 213.569,A -85,B 0,C 180,E1 -861.73,E2 -861.73} C_VEL
LIN {X 0,Y 601.38,Z 213.573,A -85,B 0,C 180,E1 -864.245,E2 -864.245} C_VEL
LIN {X 0,Y 601.407,Z 213.572,A -85,B 0,C 180,E1 -866.685,E2 -866.685} C_VEL
LIN {X 0,Y 601.394,Z 213.569,A -85,B 0,C 180,E1 -869.056,E2 -869.056} C_VEL
LIN {X 0,Y 601.415,Z 213.569,A -85,B 0,C 180,E1 -871.372,E2 -871.372} C_VEL
LIN {X 0,Y 601.419,Z 213.566,A -85,B 0,C 180,E1 -874.382,E2 -874.382} C_VEL
LIN {X 0,Y 601.399,Z 213.57,A -85,B 0,C 180,E1 -876.589,E2 -876.589} C_VEL
LIN {X 0,Y 601.421,Z 213.566,A -85,B 0,C 180,E1 -879.478,E2 -879.478} C_VEL
LIN {X 0,Y 601.388,Z 213.577,A -85,B 0,C 180,E1 -882.311,E2 -882.311} C_VEL
LIN {X 0,Y 601.392,Z 213.574,A -85,B 0,C 180,E1 -884.408,E2 -884.408} C_VEL
LIN {X 0,Y 601.384,Z 213.571,A -85,B 0,C 180,E1 -886.483,E2 -886.483} C_VEL
LIN {X 0,Y 601.39,Z 213.573,A -85,B 0,C 180,E1 -889.223,E2 -889.223} C_VEL
LIN {X 0,Y 601.412,Z 213.567,A -85,B 0,C 180,E1 -891.939,E2 -891.939} C_VEL
LIN {X 0,Y 601.404,Z 213.568,A -85,B 0,C 180,E1 -893.963,E2 -893.963} C_VEL
LIN {X 0,Y 601.43,Z 213.572,A -85,B 0,C 180,E1 -896.651,E2 -896.651} C_VEL
LIN {X 0,Y 601.448,Z 213.562,A -85,B 0,C 180,E1 -899.331,E2 -899.331} C_VEL
LIN {X 0,Y 601.431,Z 213.571,A -85,B 0,C 180,E1 -902.009,E2 -902.009} C_VEL
LIN {X 0,Y 601.385,Z 213.57,A -85,B 0,C 180,E1 -904.692,E2 -904.692} C_VEL
LIN {X 0,Y 601.402,Z 213.574,A -85,B 0,C 180,E1 -907.386,E2 -907.386} C_VEL
LIN {X 0,Y 601.387,Z 213.57,A -85,B 0,C 180,E1 -910.096,E2 -910.096} C_VEL
LIN {X 0,Y 601.403,Z 213.57,A -85,B 0,C 180,E1 -912.322,E2 -912.322} C_VEL
LIN {X 0,Y 600.744,Z 213.654,A -85,B 0,C 180,E1 -912.882,E2 -912.882} C_VEL
LIN {X 0,Y 597.903,Z 214.005,A -85,B 0,C 180,E1 -913.79,E2 -913.79} C_VEL
LIN {X 0,Y 595.495,Z 214.31,A -85,B 0,C 180,E1 -914.52,E2 -914.52} C_VEL
LIN {X 0,Y 594.454,Z 214.434,A -85,B 0,C 180,E1 -915.083,E2 -915.083} C_VEL
LIN {X 0,Y 594.366,Z 214.445,A -85,B 0,C 180,E1 -915.274,E2 -915.274} C_VEL
LIN {X 0,Y 594.357,Z 214.454,A -85,B 0,C 180,E1 -917.905,E2 -917.905} C_VEL
LIN {X 0,Y 594.4,Z 214.441,A -85,B 0,C 180,E1 -920.776,E2 -920.776} C_VEL
LIN {X 0,Y 594.348,Z 214.448,A -85,B 0,C 180,E1 -923.706,E2 -923.706} C_VEL
LIN {X 0,Y 594.348,Z 214.454,A -85,B 0,C 180,E1 -926.702,E2 -926.702} C_VEL
LIN {X 0,Y 594.379,Z 214.445,A -85,B 0,C 180,E1 -928.999,E2 -928.999} C_VEL
LIN {X 0,Y 594.377,Z 214.445,A -85,B 0,C 180,E1 -931.641,E2 -931.641} C_VEL
LIN {X 0,Y 594.38,Z 214.443,A -85,B 0,C 180,E1 -934.58,E2 -934.58} C_VEL
LIN {X 0,Y 594.394,Z 214.446,A -85,B 0,C 180,E1 -937.608,E2 -937.608} C_VEL
LIN {X 0,Y 594.369,Z 214.447,A -85,B 0,C 180,E1 -940.567,E2 -940.567} C_VEL
LIN {X 0,Y 594.355,Z 214.447,A -85,B 0,C 180,E1 -943.301,E2 -943.301} C_VEL
LIN {X 0,Y 594.339,Z 214.455,A -85,B 0,C 180,E1 -946.164,E2 -946.164} C_VEL
LIN {X 0,Y 594.362,Z 214.447,A -85,B 0,C 180,E1 -948.534,E2 -948.534} C_VEL
LIN {X 0,Y 594.372,Z 214.448,A -85,B 0,C 180,E1 -951.298,E2 -951.298} C_VEL
LIN {X 0,Y 594.357,Z 214.449,A -85,B 0,C 180,E1 -953.755,E2 -953.755} C_VEL
LIN {X 0,Y 594.371,Z 214.444,A -85,B 0,C 180,E1 -956.237,E2 -956.237} C_VEL
LIN {X 0,Y 594.327,Z 214.457,A -85,B 0,C 180,E1 -958.646,E2 -958.646} C_VEL
LIN {X 0,Y 594.318,Z 215.227,A -85,B 0,C 180,E1 -959.684,E2 -959.684} C_VEL
LIN {X 0,Y 594.269,Z 218.578,A -85,B 0,C 180,E1 -962.533,E2 -962.533} C_VEL
LIN {X 0,Y 594.262,Z 221.224,A -85,B 0,C 180,E1 -964.801,E2 -964.801} C_VEL
LIN {X 0,Y 594.242,Z 224.699,A -85,B 0,C 180,E1 -967.761,E2 -967.761} C_VEL
LIN {X 0,Y 594.208,Z 227.392,A -85,B 0,C 180,E1 -969.939,E2 -969.939} C_VEL
LIN {X 0,Y 594.193,Z 230.198,A -85,B 0,C 180,E1 -972.089,E2 -972.089} C_VEL
LIN {X 0,Y 594.229,Z 233.012,A -85,B 0,C 180,E1 -974.214,E2 -974.214} C_VEL
LIN {X 0,Y 594.231,Z 236.777,A -85,B 0,C 180,E1 -977.013,E2 -977.013} C_VEL
LIN {X 0,Y 594.208,Z 240.557,A -85,B 0,C 180,E1 -979.78,E2 -979.78} C_VEL
LIN {X 0,Y 594.219,Z 243.667,A -85,B 0,C 180,E1 -982.032,E2 -982.032} C_VEL
LIN {X 0,Y 594.651,Z 248.216,A -85,B 0,C 180,E1 -982.145,E2 -982.145} C_VEL
LIN {X 0,Y 594.595,Z 260.852,A -85,B 0,C 180,E1 -982.486,E2 -982.486} C_VEL
LIN {X 0,Y 594.579,Z 273.115,A -85,B 0,C 180,E1 -982.955,E2 -982.955} C_VEL
LIN {X 0,Y 594.478,Z 284.623,A -85,B 0,C 180,E1 -983.533,E2 -983.533} C_VEL
LIN {X 0,Y 594.462,Z 295.539,A -85,B 0,C 180,E1 -984.232,E2 -984.232} C_VEL
LIN {X 0,Y 594.399,Z 306.163,A -85,B 0,C 180,E1 -985.081,E2 -985.081} C_VEL
LIN {X 0,Y 594.348,Z 314.824,A -85,B 0,C 180,E1 -985.931,E2 -985.931} C_VEL
LIN {X 0,Y 594.319,Z 323.262,A -85,B 0,C 180,E1 -986.949,E2 -986.949} C_VEL
LIN {X 0,Y 594.267,Z 330.049,A -85,B 0,C 180,E1 -987.966,E2 -987.966} C_VEL
LIN {X 0,Y 594.29,Z 335.489,A -85,B 0,C 180,E1 -988.983,E2 -988.983} C_VEL
LIN {X 0,Y 594.26,Z 339.761,A -85,B 0,C 180,E1 -989.999,E2 -989.999} C_VEL
LIN {X 0,Y 594.242,Z 342.025,A -85,B 0,C 180,E1 -990.677,E2 -990.677} C_VEL
LIN {X 0,Y 594.248,Z 343.86,A -85,B 0,C 180,E1 -991.354,E2 -991.354} C_VEL
LIN {X 0,Y 594.241,Z 345.236,A -85,B 0,C 180,E1 -992.032,E2 -992.032} C_VEL
LIN {X 0,Y 594.258,Z 346.799,A -85,B 0,C 180,E1 -993.389,E2 -993.389} C_VEL
LIN {X 0,Y 594.255,Z 346.999,A -85,B 0,C 180,E1 -994.068,E2 -994.068} C_VEL
LIN {X 0,Y 594.252,Z 346.153,A -85,B 0,C 180,E1 -995.428,E2 -995.428} C_VEL
LIN {X 0,Y 594.26,Z 344.215,A -85,B 0,C 180,E1 -996.571,E2 -996.571} C_VEL
LIN {X 0,Y 594.244,Z 340.758,A -85,B 0,C 180,E1 -997.816,E2 -997.816} C_VEL
LIN {X 0,Y 594.253,Z 336.737,A -85,B 0,C 180,E1 -998.843,E2 -998.843} C_VEL
LIN {X 0,Y 594.287,Z 330.521,A -85,B 0,C 180,E1 -1000.045,E2 -1000.045} C_VEL
LIN {X 0,Y 594.332,Z 323.975,A -85,B 0,C 180,E1 -1001.043,E2 -1001.043} C_VEL
LIN {X 0,Y 594.38,Z 315.249,A -85,B 0,C 180,E1 -1002.114,E2 -1002.114} C_VEL
LIN {X 0,Y 594.386,Z 306.471,A -85,B 0,C 180,E1 -1002.982,E2 -1002.982} C_VEL
LIN {X 0,Y 594.446,Z 296.411,A -85,B 0,C 180,E1 -1003.795,E2 -1003.795} C_VEL
LIN {X 0,Y 594.497,Z 286.27,A -85,B 0,C 180,E1 -1004.461,E2 -1004.461} C_VEL
LIN {X 0,Y 594.555,Z 274.564,A -85,B 0,C 180,E1 -1005.072,E2 -1005.072} C_VEL
LIN {X 0,Y 594.583,Z 262.366,A -85,B 0,C 180,E1 -1005.554,E2 -1005.554} C_VEL
LIN {X 0,Y 594.648,Z 249.039,A -85,B 0,C 180,E1 -1005.926,E2 -1005.926} C_VEL
LIN {X 0,Y 594.235,Z 243.68,A -85,B 0,C 180,E1 -1006.048,E2 -1006.048} C_VEL
LIN {X 0,Y 594.24,Z 239.763,A -85,B 0,C 180,E1 -1008.888,E2 -1008.888} C_VEL
LIN {X 0,Y 594.217,Z 236.195,A -85,B 0,C 180,E1 -1011.508,E2 -1011.508} C_VEL
LIN {X 0,Y 594.232,Z 233.234,A -85,B 0,C 180,E1 -1013.709,E2 -1013.709} C_VEL
LIN {X 0,Y 594.223,Z 230.212,A -85,B 0,C 180,E1 -1015.99,E2 -1015.99} C_VEL
LIN {X 0,Y 594.247,Z 227.284,A -85,B 0,C 180,E1 -1018.232,E2 -1018.232} C_VEL
LIN {X 0,Y 594.252,Z 224.4,A -85,B 0,C 180,E1 -1020.566,E2 -1020.566} C_VEL
LIN {X 0,Y 594.285,Z 221.692,A -85,B 0,C 180,E1 -1022.955,E2 -1022.955} C_VEL
LIN {X 0,Y 594.287,Z 218.778,A -85,B 0,C 180,E1 -1025.412,E2 -1025.412} C_VEL
LIN {X 0,Y 594.293,Z 215.785,A -85,B 0,C 180,E1 -1027.946,E2 -1027.946} C_VEL
LIN {X 0,Y 594.294,Z 214.776,A -85,B 0,C 180,E1 -1028.81,E2 -1028.81} C_VEL
LIN {X 0,Y 594.365,Z 214.447,A -85,B 0,C 180,E1 -1030.566,E2 -1030.566} C_VEL
LIN {X 0,Y 594.361,Z 214.447,A -85,B 0,C 180,E1 -1033.298,E2 -1033.298} C_VEL
LIN {X 0,Y 594.345,Z 214.453,A -85,B 0,C 180,E1 -1036.161,E2 -1036.161} C_VEL
LIN {X 0,Y 594.358,Z 214.447,A -85,B 0,C 180,E1 -1038.534,E2 -1038.534} C_VEL
LIN {X 0,Y 594.379,Z 214.446,A -85,B 0,C 180,E1 -1041.294,E2 -1041.294} C_VEL
LIN {X 0,Y 594.39,Z 214.444,A -85,B 0,C 180,E1 -1043.758,E2 -1043.758} C_VEL
LIN {X 0,Y 594.355,Z 214.449,A -85,B 0,C 180,E1 -1046.237,E2 -1046.237} C_VEL
LIN {X 0,Y 594.353,Z 214.448,A -85,B 0,C 180,E1 -1048.648,E2 -1048.648} C_VEL
LIN {X 0,Y 594.375,Z 214.448,A -85,B 0,C 180,E1 -1051.041,E2 -1051.041} C_VEL
LIN {X 0,Y 594.384,Z 214.448,A -85,B 0,C 180,E1 -1053.975,E2 -1053.975} C_VEL
LIN {X 0,Y 594.381,Z 214.445,A -85,B 0,C 180,E1 -1056.295,E2 -1056.295} C_VEL
LIN {X 0,Y 594.385,Z 214.448,A -85,B 0,C 180,E1 -1059.224,E2 -1059.224} C_VEL
LIN {X 0,Y 594.338,Z 214.452,A -85,B 0,C 180,E1 -1062.094,E2 -1062.094} C_VEL
LIN {X 0,Y 594.367,Z 214.45,A -85,B 0,C 180,E1 -1064.219,E2 -1064.219} C_VEL
LIN {X 0,Y 594.363,Z 214.449,A -85,B 0,C 180,E1 -1067.017,E2 -1067.017} C_VEL
LIN {X 0,Y 594.382,Z 214.449,A -85,B 0,C 180,E1 -1069.095,E2 -1069.095} C_VEL
LIN {X 0,Y 594.399,Z 214.443,A -85,B 0,C 180,E1 -1071.843,E2 -1071.843} C_VEL
LIN {X 0,Y 594.399,Z 214.442,A -85,B 0,C 180,E1 -1074.572,E2 -1074.572} C_VEL
LIN {X 0,Y 594.4,Z 214.447,A -85,B 0,C 180,E1 -1077.289,E2 -1077.289} C_VEL
LIN {X 0,Y 594.383,Z 214.445,A -85,B 0,C 180,E1 -1080,E2 -1080} C_VEL
LIN {X 0,Y 594.399,Z 214.442,A -85,B 0,C 180,E1 -1082.711,E2 -1082.711} C_VEL
LIN {X 0,Y 594.39,Z 214.45,A -85,B 0,C 180,E1 -1085.428,E2 -1085.428} C_VEL
LIN {X 0,Y 594.405,Z 214.441,A -85,B 0,C 180,E1 -1088.157,E2 -1088.157} C_VEL
LIN {X 0,Y 594.36,Z 214.446,A -85,B 0,C 180,E1 -1091.066,E2 -1091.066} C_VEL
LIN {X 0,Y 594.368,Z 214.452,A -85,B 0,C 180,E1 -1093.679,E2 -1093.679} C_VEL
LIN {X 0,Y 594.385,Z 214.447,A -85,B 0,C 180,E1 -1096.721,E2 -1096.721} C_VEL
LIN {X 0,Y 594.357,Z 214.446,A -85,B 0,C 180,E1 -1099.335,E2 -1099.335} C_VEL
LIN {X 0,Y 594.339,Z 214.451,A -85,B 0,C 180,E1 -1101.504,E2 -1101.504} C_VEL
LIN {X 0,Y 594.378,Z 214.444,A -85,B 0,C 180,E1 -1104.447,E2 -1104.447} C_VEL
LIN {X 0,Y 594.381,Z 214.449,A -85,B 0,C 180,E1 -1106.7,E2 -1106.7} C_VEL
LIN {X 0,Y 594.377,Z 214.445,A -85,B 0,C 180,E1 -1108.999,E2 -1108.999} C_VEL
LIN {X 0,Y 594.363,Z 214.451,A -85,B 0,C 180,E1 -1111.643,E2 -1111.643} C_VEL
LIN {X 0,Y 594.367,Z 214.447,A -85,B 0,C 180,E1 -1114.581,E2 -1114.581} C_VEL
LIN {X 0,Y 594.384,Z 214.443,A -85,B 0,C 180,E1 -1117.61,E2 -1117.61} C_VEL
LIN {X 0,Y 594.362,Z 214.447,A -85,B 0,C 180,E1 -1120.568,E2 -1120.568} C_VEL
LIN {X 0,Y 594.349,Z 214.455,A -85,B 0,C 180,E1 -1123.301,E2 -1123.301} C_VEL
LIN {X 0,Y 594.36,Z 214.448,A -85,B 0,C 180,E1 -1126.162,E2 -1126.162} C_VEL
LIN {X 0,Y 594.386,Z 214.444,A -85,B 0,C 180,E1 -1129.177,E2 -1129.177} C_VEL
LIN {X 0,Y 594.375,Z 214.447,A -85,B 0,C 180,E1 -1132.06,E2 -1132.06} C_VEL
LIN {X 0,Y 594.377,Z 214.64,A -85,B 0,C 180,E1 -1133.969,E2 -1133.969} C_VEL
LIN {X 0,Y 594.613,Z 219.274,A -85,B 0,C 180,E1 -1135.437,E2 -1135.437} C_VEL
LIN {X 0,Y 594.597,Z 227.217,A -85,B 0,C 180,E1 -1137.868,E2 -1137.868} C_VEL
LIN {X 0,Y 594.562,Z 236.484,A -85,B 0,C 180,E1 -1140.625,E2 -1140.625} C_VEL
LIN {X 0,Y 594.468,Z 245.751,A -85,B 0,C 180,E1 -1143.306,E2 -1143.306} C_VEL
LIN {X 0,Y 594.445,Z 255.019,A -85,B 0,C 180,E1 -1145.929,E2 -1145.929} C_VEL
LIN {X 0,Y 594.402,Z 265.496,A -85,B 0,C 180,E1 -1148.832,E2 -1148.832} C_VEL
LIN {X 0,Y 594.374,Z 274.877,A -85,B 0,C 180,E1 -1151.383,E2 -1151.383} C_VEL
LIN {X 0,Y 594.318,Z 285.468,A -85,B 0,C 180,E1 -1154.219,E2 -1154.219} C_VEL
LIN {X 0,Y 594.278,Z 296.059,A -85,B 0,C 180,E1 -1157.016,E2 -1157.016} C_VEL
LIN {X 0,Y 594.298,Z 299.809,A -85,B 0,C 180,E1 -1157.944,E2 -1157.944} C_VEL
LIN {X 0,Y 594.681,Z 304.146,A -85,B 0,C 180,E1 -1158.022,E2 -1158.022} C_VEL
LIN {X 0,Y 594.621,Z 317.774,A -85,B 0,C 180,E1 -1158.345,E2 -1158.345} C_VEL
LIN {X 0,Y 594.547,Z 328.817,A -85,B 0,C 180,E1 -1158.727,E2 -1158.727} C_VEL
LIN {X 0,Y 594.49,Z 340.654,A -85,B 0,C 180,E1 -1159.27,E2 -1159.27} C_VEL
LIN {X 0,Y 594.463,Z 352.214,A -85,B 0,C 180,E1 -1159.958,E2 -1159.958} C_VEL
LIN {X 0,Y 594.414,Z 362.608,A -85,B 0,C 180,E1 -1160.731,E2 -1160.731} C_VEL
LIN {X 0,Y 594.382,Z 371.123,A -85,B 0,C 180,E1 -1161.502,E2 -1161.502} C_VEL
LIN {X 0,Y 594.347,Z 378.969,A -85,B 0,C 180,E1 -1162.356,E2 -1162.356} C_VEL
LIN {X 0,Y 594.282,Z 386.817,A -85,B 0,C 180,E1 -1163.409,E2 -1163.409} C_VEL
LIN {X 0,Y 594.289,Z 393.686,A -85,B 0,C 180,E1 -1164.572,E2 -1164.572} C_VEL
LIN {X 0,Y 594.27,Z 398.375,A -85,B 0,C 180,E1 -1165.592,E2 -1165.592} C_VEL
LIN {X 0,Y 594.267,Z 401.959,A -85,B 0,C 180,E1 -1166.611,E2 -1166.611} C_VEL
LIN {X 0,Y 594.226,Z 403.811,A -85,B 0,C 180,E1 -1167.289,E2 -1167.289} C_VEL
LIN {X 0,Y 594.242,Z 405.203,A -85,B 0,C 180,E1 -1167.968,E2 -1167.968} C_VEL
LIN {X 0,Y 594.239,Z 406.784,A -85,B 0,C 180,E1 -1169.323,E2 -1169.323} C_VEL
LIN {X 0,Y 594.236,Z 407,A -85,B 0,C 180,E1 -1170.001,E2 -1170.001} C_VEL
LIN {X 0,Y 594.247,Z 406.183,A -85,B 0,C 180,E1 -1171.356,E2 -1171.356} C_VEL
LIN {X 0,Y 594.242,Z 405.2,A -85,B 0,C 180,E1 -1172.034,E2 -1172.034} C_VEL
LIN {X 0,Y 594.226,Z 403.807,A -85,B 0,C 180,E1 -1172.713,E2 -1172.713} C_VEL
LIN {X 0,Y 594.289,Z 400.893,A -85,B 0,C 180,E1 -1173.73,E2 -1173.73} C_VEL
LIN {X 0,Y 594.241,Z 396.946,A -85,B 0,C 180,E1 -1174.75,E2 -1174.75} C_VEL
LIN {X 0,Y 594.305,Z 390.871,A -85,B 0,C 180,E1 -1175.94,E2 -1175.94} C_VEL
LIN {X 0,Y 594.309,Z 384.229,A -85,B 0,C 180,E1 -1176.963,E2 -1176.963} C_VEL
LIN {X 0,Y 594.36,Z 375.981,A -85,B 0,C 180,E1 -1177.987,E2 -1177.987} C_VEL
LIN {X 0,Y 594.382,Z 367.526,A -85,B 0,C 180,E1 -1178.843,E2 -1178.843} C_VEL
LIN {X 0,Y 594.432,Z 357.079,A -85,B 0,C 180,E1 -1179.7,E2 -1179.7} C_VEL
LIN {X 0,Y 594.45,Z 346.741,A -85,B 0,C 180,E1 -1180.388,E2 -1180.388} C_VEL
LIN {X 0,Y 594.5,Z 334.76,A -85,B 0,C 180,E1 -1181.019,E2 -1181.019} C_VEL
LIN {X 0,Y 594.561,Z 322.468,A -85,B 0,C 180,E1 -1181.506,E2 -1181.506} C_VEL
LIN {X 0,Y 594.646,Z 309.398,A -85,B 0,C 180,E1 -1181.873,E2 -1181.873} C_VEL
LIN {X 0,Y 594.596,Z 301.549,A -85,B 0,C 180,E1 -1182.025,E2 -1182.025} C_VEL
LIN {X 0,Y 594.284,Z 299.527,A -85,B 0,C 180,E1 -1182.075,E2 -1182.075} C_VEL
LIN {X 0,Y 594.305,Z 289.432,A -85,B 0,C 180,E1 -1184.73,E2 -1184.73} C_VEL
LIN {X 0,Y 594.336,Z 278.841,A -85,B 0,C 180,E1 -1187.551,E2 -1187.551} C_VEL
LIN {X 0,Y 594.383,Z 268.25,A -85,B 0,C 180,E1 -1190.415,E2 -1190.415} C_VEL
LIN {X 0,Y 594.441,Z 257.659,A -85,B 0,C 180,E1 -1193.333,E2 -1193.333} C_VEL
LIN {X 0,Y 594.488,Z 248.031,A -85,B 0,C 180,E1 -1196.042,E2 -1196.042} C_VEL
LIN {X 0,Y 594.488,Z 239.145,A -85,B 0,C 180,E1 -1198.601,E2 -1198.601} C_VEL
LIN {X 0,Y 594.589,Z 229.857,A -85,B 0,C 180,E1 -1201.338,E2 -1201.338} C_VEL
LIN {X 0,Y 594.615,Z 221.914,A -85,B 0,C 180,E1 -1203.747,E2 -1203.747} C_VEL
LIN {X 0,Y 594.484,Z 215.294,A -85,B 0,C 180,E1 -1205.817,E2 -1205.817} C_VEL
LIN {X 0,Y 594.346,Z 214.453,A -85,B 0,C 180,E1 -1206.141,E2 -1206.141} C_VEL
LIN {X 0,Y 594.367,Z 214.452,A -85,B 0,C 180,E1 -1208.807,E2 -1208.807} C_VEL
LIN {X 0,Y 594.38,Z 214.446,A -85,B 0,C 180,E1 -1211.848,E2 -1211.848} C_VEL
LIN {X 0,Y 594.371,Z 214.444,A -85,B 0,C 180,E1 -1214.809,E2 -1214.809} C_VEL
LIN {X 0,Y 594.373,Z 214.452,A -85,B 0,C 180,E1 -1217.625,E2 -1217.625} C_VEL
LIN {X 0,Y 594.375,Z 214.443,A -85,B 0,C 180,E1 -1220.319,E2 -1220.319} C_VEL
LIN {X 0,Y 594.384,Z 214.45,A -85,B 0,C 180,E1 -1222.913,E2 -1222.913} C_VEL
LIN {X 0,Y 594.362,Z 214.45,A -85,B 0,C 180,E1 -1226.238,E2 -1226.238} C_VEL
LIN {X 0,Y 594.363,Z 214.447,A -85,B 0,C 180,E1 -1228.649,E2 -1228.649} C_VEL
LIN {X 0,Y 594.38,Z 214.443,A -85,B 0,C 180,E1 -1231.044,E2 -1231.044} C_VEL
LIN {X 0,Y 594.378,Z 214.445,A -85,B 0,C 180,E1 -1234.056,E2 -1234.056} C_VEL
LIN {X 0,Y 594.38,Z 214.443,A -85,B 0,C 180,E1 -1236.295,E2 -1236.295} C_VEL
LIN {X 0,Y 594.397,Z 214.444,A -85,B 0,C 180,E1 -1239.224,E2 -1239.224} C_VEL
LIN {X 0,Y 594.34,Z 214.451,A -85,B 0,C 180,E1 -1242.095,E2 -1242.095} C_VEL
LIN {X 0,Y 594.345,Z 214.455,A -85,B 0,C 180,E1 -1244.218,E2 -1244.218} C_VEL
LIN {X 0,Y 594.355,Z 214.449,A -85,B 0,C 180,E1 -1246.32,E2 -1246.32} C_VEL
LIN {X 0,Y 594.35,Z 214.449,A -85,B 0,C 180,E1 -1249.094,E2 -1249.094} C_VEL
LIN {X 0,Y 594.365,Z 214.446,A -85,B 0,C 180,E1 -1251.843,E2 -1251.843} C_VEL
LIN {X 0,Y 594.392,Z 214.446,A -85,B 0,C 180,E1 -1254.572,E2 -1254.572} C_VEL
LIN {X 0,Y 594.411,Z 214.439,A -85,B 0,C 180,E1 -1257.289,E2 -1257.289} C_VEL
LIN {X 0,Y 594.421,Z 214.444,A -85,B 0,C 180,E1 -1260,E2 -1260} C_VEL
LIN {X 0,Y 594.385,Z 214.442,A -85,B 0,C 180,E1 -1262.711,E2 -1262.711} C_VEL
LIN {X 0,Y 594.383,Z 214.45,A -85,B 0,C 180,E1 -1265.428,E2 -1265.428} C_VEL
LIN {X 0,Y 594.343,Z 214.447,A -85,B 0,C 180,E1 -1268.158,E2 -1268.158} C_VEL
LIN {X 0,Y 594.393,Z 214.445,A -85,B 0,C 180,E1 -1271.072,E2 -1271.072} C_VEL
LIN {X 0,Y 594.374,Z 214.444,A -85,B 0,C 180,E1 -1273.679,E2 -1273.679} C_VEL
LIN {X 0,Y 594.366,Z 214.445,A -85,B 0,C 180,E1 -1275.274,E2 -1275.274} C_VEL
LIN {X 0,Y 593.688,Z 214.535,A -85,B 0,C 180,E1 -1275.84,E2 -1275.84} C_VEL
LIN {X 0,Y 590.823,Z 214.893,A -85,B 0,C 180,E1 -1276.758,E2 -1276.758} C_VEL
LIN {X 0,Y 588.415,Z 215.194,A -85,B 0,C 180,E1 -1277.496,E2 -1277.496} C_VEL
LIN {X 0,Y 587.391,Z 215.319,A -85,B 0,C 180,E1 -1278.066,E2 -1278.066} C_VEL
LIN {X 0,Y 587.312,Z 215.326,A -85,B 0,C 180,E1 -1278.259,E2 -1278.259} C_VEL
LIN {X 0,Y 587.339,Z 215.323,A -85,B 0,C 180,E1 -1281.037,E2 -1281.037} C_VEL
LIN {X 0,Y 587.288,Z 215.326,A -85,B 0,C 180,E1 -1284.009,E2 -1284.009} C_VEL
LIN {X 0,Y 587.287,Z 215.328,A -85,B 0,C 180,E1 -1286.281,E2 -1286.281} C_VEL
LIN {X 0,Y 587.348,Z 215.32,A -85,B 0,C 180,E1 -1289.132,E2 -1289.132} C_VEL
LIN {X 0,Y 587.346,Z 215.324,A -85,B 0,C 180,E1 -1291.834,E2 -1291.834} C_VEL
LIN {X 0,Y 587.347,Z 215.321,A -85,B 0,C 180,E1 -1294.346,E2 -1294.346} C_VEL
LIN {X 0,Y 587.349,Z 215.324,A -85,B 0,C 180,E1 -1297.608,E2 -1297.608} C_VEL
LIN {X 0,Y 587.315,Z 215.323,A -85,B 0,C 180,E1 -1300.255,E2 -1300.255} C_VEL
LIN {X 0,Y 587.31,Z 215.328,A -85,B 0,C 180,E1 -1303.007,E2 -1303.007} C_VEL
LIN {X 0,Y 587.291,Z 215.331,A -85,B 0,C 180,E1 -1306.045,E2 -1306.045} C_VEL
LIN {X 0,Y 587.292,Z 215.325,A -85,B 0,C 180,E1 -1308.93,E2 -1308.93} C_VEL
LIN {X 0,Y 587.323,Z 215.329,A -85,B 0,C 180,E1 -1311.519,E2 -1311.519} C_VEL
LIN {X 0,Y 587.297,Z 215.325,A -85,B 0,C 180,E1 -1314.099,E2 -1314.099} C_VEL
LIN {X 0,Y 587.343,Z 215.327,A -85,B 0,C 180,E1 -1316.888,E2 -1316.888} C_VEL
LIN {X 0,Y 587.234,Z 215.341,A -85,B 0,C 180,E1 -1319.027,E2 -1319.027} C_VEL
LIN {X 0,Y 587.211,Z 217.885,A -85,B 0,C 180,E1 -1321.396,E2 -1321.396} C_VEL
LIN {X 0,Y 587.177,Z 221.442,A -85,B 0,C 180,E1 -1324.475,E2 -1324.475} C_VEL
LIN {X 0,Y 587.194,Z 224.983,A -85,B 0,C 180,E1 -1327.479,E2 -1327.479} C_VEL
LIN {X 0,Y 587.157,Z 227.511,A -85,B 0,C 180,E1 -1329.688,E2 -1329.688} C_VEL
LIN {X 0,Y 587.117,Z 230.27,A -85,B 0,C 180,E1 -1331.866,E2 -1331.866} C_VEL
LIN {X 0,Y 587.141,Z 233.083,A -85,B 0,C 180,E1 -1334.019,E2 -1334.019} C_VEL
LIN {X 0,Y 587.13,Z 236.848,A -85,B 0,C 180,E1 -1336.853,E2 -1336.853} C_VEL
LIN {X 0,Y 587.123,Z 240.626,A -85,B 0,C 180,E1 -1339.655,E2 -1339.655} C_VEL
LIN {X 0,Y 587.14,Z 243.676,A -85,B 0,C 180,E1 -1341.892,E2 -1341.892} C_VEL
LIN {X 0,Y 587.71,Z 249.38,A -85,B 0,C 180,E1 -1342.03,E2 -1342.03} C_VEL
LIN {X 0,Y 587.649,Z 262.309,A -85,B 0,C 180,E1 -1342.396,E2 -1342.396} C_VEL
LIN {X 0,Y 587.606,Z 274.228,A -85,B 0,C 180,E1 -1342.871,E2 -1342.871} C_VEL
LIN {X 0,Y 587.478,Z 285.724,A -85,B 0,C 180,E1 -1343.47,E2 -1343.47} C_VEL
LIN {X 0,Y 587.427,Z 297.357,A -85,B 0,C 180,E1 -1344.248,E2 -1344.248} C_VEL
LIN {X 0,Y 587.364,Z 306.714,A -85,B 0,C 180,E1 -1345.022,E2 -1345.022} C_VEL
LIN {X 0,Y 587.297,Z 315.283,A -85,B 0,C 180,E1 -1345.882,E2 -1345.882} C_VEL
LIN {X 0,Y 587.257,Z 323.614,A -85,B 0,C 180,E1 -1346.912,E2 -1346.912} C_VEL
LIN {X 0,Y 587.178,Z 330.338,A -85,B 0,C 180,E1 -1347.941,E2 -1347.941} C_VEL
LIN {X 0,Y 587.203,Z 335.718,A -85,B 0,C 180,E1 -1348.97,E2 -1348.97} C_VEL
LIN {X 0,Y 587.163,Z 339.937,A -85,B 0,C 180,E1 -1349.999,E2 -1349.999} C_VEL
LIN {X 0,Y 587.143,Z 342.176,A -85,B 0,C 180,E1 -1350.685,E2 -1350.685} C_VEL
LIN {X 0,Y 587.148,Z 343.968,A -85,B 0,C 180,E1 -1351.371,E2 -1351.371} C_VEL
LIN {X 0,Y 587.14,Z 345.315,A -85,B 0,C 180,E1 -1352.057,E2 -1352.057} C_VEL
LIN {X 0,Y 587.181,Z 346.832,A -85,B 0,C 180,E1 -1353.43,E2 -1353.43} C_VEL
LIN {X 0,Y 587.17,Z 346.99,A -85,B 0,C 180,E1 -1354.117,E2 -1354.117} C_VEL
LIN {X 0,Y 587.17,Z 346.097,A -85,B 0,C 180,E1 -1355.494,E2 -1355.494} C_VEL
LIN {X 0,Y 587.187,Z 344.276,A -85,B 0,C 180,E1 -1356.573,E2 -1356.573} C_VEL
LIN {X 0,Y 587.172,Z 340.585,A -85,B 0,C 180,E1 -1357.911,E2 -1357.911} C_VEL
LIN {X 0,Y 587.159,Z 336.512,A -85,B 0,C 180,E1 -1358.951,E2 -1358.951} C_VEL
LIN {X 0,Y 587.215,Z 330.229,A -85,B 0,C 180,E1 -1360.167,E2 -1360.167} C_VEL
LIN {X 0,Y 587.265,Z 323.492,A -85,B 0,C 180,E1 -1361.195,E2 -1361.195} C_VEL
LIN {X 0,Y 587.328,Z 316.344,A -85,B 0,C 180,E1 -1362.086,E2 -1362.086} C_VEL
LIN {X 0,Y 587.343,Z 307.86,A -85,B 0,C 180,E1 -1362.964,E2 -1362.964} C_VEL
LIN {X 0,Y 587.421,Z 297.339,A -85,B 0,C 180,E1 -1363.843,E2 -1363.843} C_VEL
LIN {X 0,Y 587.49,Z 286.887,A -85,B 0,C 180,E1 -1364.548,E2 -1364.548} C_VEL
LIN {X 0,Y 587.578,Z 275.387,A -85,B 0,C 180,E1 -1365.167,E2 -1365.167} C_VEL
LIN {X 0,Y 587.616,Z 263.497,A -85,B 0,C 180,E1 -1365.654,E2 -1365.654} C_VEL
LIN {X 0,Y 587.695,Z 250.638,A -85,B 0,C 180,E1 -1366.03,E2 -1366.03} C_VEL
LIN {X 0,Y 587.393,Z 245.365,A -85,B 0,C 180,E1 -1366.15,E2 -1366.15} C_VEL
LIN {X 0,Y 587.139,Z 243.67,A -85,B 0,C 180,E1 -1366.202,E2 -1366.202} C_VEL
LIN {X 0,Y 587.149,Z 239.881,A -85,B 0,C 180,E1 -1368.983,E2 -1368.983} C_VEL
LIN {X 0,Y 587.135,Z 236.121,A -85,B 0,C 180,E1 -1371.78,E2 -1371.78} C_VEL
LIN {X 0,Y 587.157,Z 232.17,A -85,B 0,C 180,E1 -1374.766,E2 -1374.766} C_VEL
LIN {X 0,Y 587.155,Z 228.42,A -85,B 0,C 180,E1 -1377.655,E2 -1377.655} C_VEL
LIN {X 0,Y 587.206,Z 225.109,A -85,B 0,C 180,E1 -1380.487,E2 -1380.487} C_VEL
LIN {X 0,Y 587.202,Z 221.764,A -85,B 0,C 180,E1 -1383.404,E2 -1383.404} C_VEL
LIN {X 0,Y 587.211,Z 218.83,A -85,B 0,C 180,E1 -1385.904,E2 -1385.904} C_VEL
LIN {X 0,Y 587.243,Z 215.34,A -85,B 0,C 180,E1 -1388.93,E2 -1388.93} C_VEL
LIN {X 0,Y 587.333,Z 215.327,A -85,B 0,C 180,E1 -1391.155,E2 -1391.155} C_VEL
LIN {X 0,Y 587.321,Z 215.327,A -85,B 0,C 180,E1 -1394.112,E2 -1394.112} C_VEL
LIN {X 0,Y 587.296,Z 215.327,A -85,B 0,C 180,E1 -1396.991,E2 -1396.991} C_VEL
LIN {X 0,Y 587.304,Z 215.327,A -85,B 0,C 180,E1 -1399.744,E2 -1399.744} C_VEL
LIN {X 0,Y 587.339,Z 215.325,A -85,B 0,C 180,E1 -1402.392,E2 -1402.392} C_VEL
LIN {X 0,Y 587.34,Z 215.321,A -85,B 0,C 180,E1 -1404.945,E2 -1404.945} C_VEL
LIN {X 0,Y 587.33,Z 215.327,A -85,B 0,C 180,E1 -1407.42,E2 -1407.42} C_VEL
LIN {X 0,Y 587.306,Z 215.325,A -85,B 0,C 180,E1 -1409.828,E2 -1409.828} C_VEL
LIN {X 0,Y 587.343,Z 215.325,A -85,B 0,C 180,E1 -1412.306,E2 -1412.306} C_VEL
LIN {X 0,Y 587.331,Z 215.324,A -85,B 0,C 180,E1 -1414.483,E2 -1414.483} C_VEL
LIN {X 0,Y 587.308,Z 215.328,A -85,B 0,C 180,E1 -1417.131,E2 -1417.131} C_VEL
LIN {X 0,Y 587.309,Z 215.325,A -85,B 0,C 180,E1 -1419.694,E2 -1419.694} C_VEL
LIN {X 0,Y 587.292,Z 215.328,A -85,B 0,C 180,E1 -1421.872,E2 -1421.872} C_VEL
LIN {X 0,Y 587.323,Z 215.33,A -85,B 0,C 180,E1 -1424.025,E2 -1424.025} C_VEL
LIN {X 0,Y 587.352,Z 215.32,A -85,B 0,C 180,E1 -1426.154,E2 -1426.154} C_VEL
LIN {X 0,Y 587.382,Z 215.323,A -85,B 0,C 180,E1 -1428.963,E2 -1428.963} C_VEL
LIN {X 0,Y 587.351,Z 215.32,A -85,B 0,C 180,E1 -1431.744,E2 -1431.744} C_VEL
LIN {X 0,Y 587.364,Z 215.318,A -85,B 0,C 180,E1 -1434.507,E2 -1434.507} C_VEL
LIN {X 0,Y 587.366,Z 215.324,A -85,B 0,C 180,E1 -1437.257,E2 -1437.257} C_VEL
LIN {X 0,Y 587.353,Z 215.32,A -85,B 0,C 180,E1 -1440,E2 -1440} C_VEL
LIN {X 0,Y 587.365,Z 215.318,A -85,B 0,C 180,E1 -1442.743,E2 -1442.743} C_VEL
LIN {X 0,Y 587.354,Z 215.325,A -85,B 0,C 180,E1 -1445.493,E2 -1445.493} C_VEL
LIN {X 0,Y 587.359,Z 215.32,A -85,B 0,C 180,E1 -1448.255,E2 -1448.255} C_VEL
LIN {X 0,Y 587.336,Z 215.321,A -85,B 0,C 180,E1 -1451.134,E2 -1451.134} C_VEL
LIN {X 0,Y 587.354,Z 215.319,A -85,B 0,C 180,E1 -1454.261,E2 -1454.261} C_VEL
LIN {X 0,Y 587.351,Z 215.321,A -85,B 0,C 180,E1 -1457.406,E2 -1457.406} C_VEL
LIN {X 0,Y 587.314,Z 215.331,A -85,B 0,C 180,E1 -1460.305,E2 -1460.305} C_VEL
LIN {X 0,Y 587.3,Z 215.329,A -85,B 0,C 180,E1 -1463.26,E2 -1463.26} C_VEL
LIN {X 0,Y 587.333,Z 215.324,A -85,B 0,C 180,E1 -1465.517,E2 -1465.517} C_VEL
LIN {X 0,Y 587.341,Z 215.321,A -85,B 0,C 180,E1 -1467.818,E2 -1467.818} C_VEL
LIN {X 0,Y 587.334,Z 215.324,A -85,B 0,C 180,E1 -1470.512,E2 -1470.512} C_VEL
LIN {X 0,Y 587.324,Z 215.33,A -85,B 0,C 180,E1 -1473.397,E2 -1473.397} C_VEL
LIN {X 0,Y 587.284,Z 215.328,A -85,B 0,C 180,E1 -1475.901,E2 -1475.901} C_VEL
LIN {X 0,Y 587.325,Z 215.328,A -85,B 0,C 180,E1 -1478.48,E2 -1478.48} C_VEL
LIN {X 0,Y 587.329,Z 215.323,A -85,B 0,C 180,E1 -1481.158,E2 -1481.158} C_VEL
LIN {X 0,Y 587.303,Z 215.326,A -85,B 0,C 180,E1 -1484.113,E2 -1484.113} C_VEL
LIN {X 0,Y 587.309,Z 215.327,A -85,B 0,C 180,E1 -1486.995,E2 -1486.995} C_VEL
LIN {X 0,Y 587.324,Z 215.329,A -85,B 0,C 180,E1 -1489.748,E2 -1489.748} C_VEL
LIN {X 0,Y 587.336,Z 215.323,A -85,B 0,C 180,E1 -1492.393,E2 -1492.393} C_VEL
LIN {X 0,Y 587.334,Z 215.467,A -85,B 0,C 180,E1 -1493.733,E2 -1493.733} C_VEL
LIN {X 0,Y 587.658,Z 220.421,A -85,B 0,C 180,E1 -1495.33,E2 -1495.33} C_VEL
LIN {X 0,Y 587.639,Z 228.457,A -85,B 0,C 180,E1 -1497.821,E2 -1497.821} C_VEL
LIN {X 0,Y 587.533,Z 238.492,A -85,B 0,C 180,E1 -1500.835,E2 -1500.835} C_VEL
LIN {X 0,Y 587.475,Z 247.075,A -85,B 0,C 180,E1 -1503.346,E2 -1503.346} C_VEL
LIN {X 0,Y 587.419,Z 256.342,A -85,B 0,C 180,E1 -1505.998,E2 -1505.998} C_VEL
LIN {X 0,Y 587.357,Z 265.611,A -85,B 0,C 180,E1 -1508.597,E2 -1508.597} C_VEL
LIN {X 0,Y 587.319,Z 276.201,A -85,B 0,C 180,E1 -1511.513,E2 -1511.513} C_VEL
LIN {X 0,Y 587.257,Z 286.792,A -85,B 0,C 180,E1 -1514.38,E2 -1514.38} C_VEL
LIN {X 0,Y 587.203,Z 297.383,A -85,B 0,C 180,E1 -1517.209,E2 -1517.209} C_VEL
LIN {X 0,Y 587.211,Z 299.576,A -85,B 0,C 180,E1 -1517.791,E2 -1517.791} C_VEL
LIN {X 0,Y 587.737,Z 304.146,A -85,B 0,C 180,E1 -1517.878,E2 -1517.878} C_VEL
LIN {X 0,Y 587.67,Z 317.775,A -85,B 0,C 180,E1 -1518.205,E2 -1518.205} C_VEL
LIN {X 0,Y 587.562,Z 330.451,A -85,B 0,C 180,E1 -1518.658,E2 -1518.658} C_VEL
LIN {X 0,Y 587.49,Z 342.228,A -85,B 0,C 180,E1 -1519.228,E2 -1519.228} C_VEL
LIN {X 0,Y 587.456,Z 353.492,A -85,B 0,C 180,E1 -1519.924,E2 -1519.924} C_VEL
LIN {X 0,Y 587.384,Z 363.659,A -85,B 0,C 180,E1 -1520.706,E2 -1520.706} C_VEL
LIN {X 0,Y 587.339,Z 372.797,A -85,B 0,C 180,E1 -1521.572,E2 -1521.572} C_VEL
LIN {X 0,Y 587.258,Z 381.699,A -85,B 0,C 180,E1 -1522.609,E2 -1522.609} C_VEL
LIN {X 0,Y 587.195,Z 388.747,A -85,B 0,C 180,E1 -1523.627,E2 -1523.627} C_VEL
LIN {X 0,Y 587.211,Z 393.686,A -85,B 0,C 180,E1 -1524.507,E2 -1524.507} C_VEL
LIN {X 0,Y 587.188,Z 398.375,A -85,B 0,C 180,E1 -1525.539,E2 -1525.539} C_VEL
LIN {X 0,Y 587.193,Z 401.959,A -85,B 0,C 180,E1 -1526.57,E2 -1526.57} C_VEL
LIN {X 0,Y 587.132,Z 403.811,A -85,B 0,C 180,E1 -1527.257,E2 -1527.257} C_VEL
LIN {X 0,Y 587.141,Z 405.203,A -85,B 0,C 180,E1 -1527.943,E2 -1527.943} C_VEL
LIN {X 0,Y 587.14,Z 406.785,A -85,B 0,C 180,E1 -1529.315,E2 -1529.315} C_VEL
LIN {X 0,Y 587.137,Z 407,A -85,B 0,C 180,E1 -1530.001,E2 -1530.001} C_VEL
LIN {X 0,Y 587.147,Z 406.183,A -85,B 0,C 180,E1 -1531.373,E2 -1531.373} C_VEL
LIN {X 0,Y 587.141,Z 405.2,A -85,B 0,C 180,E1 -1532.059,E2 -1532.059} C_VEL
LIN {X 0,Y 587.132,Z 403.807,A -85,B 0,C 180,E1 -1532.745,E2 -1532.745} C_VEL
LIN {X 0,Y 587.213,Z 400.893,A -85,B 0,C 180,E1 -1533.775,E2 -1533.775} C_VEL
LIN {X 0,Y 587.147,Z 396.946,A -85,B 0,C 180,E1 -1534.807,E2 -1534.807} C_VEL
LIN {X 0,Y 587.218,Z 390.871,A -85,B 0,C 180,E1 -1536.012,E2 -1536.012} C_VEL
LIN {X 0,Y 587.246,Z 384.229,A -85,B 0,C 180,E1 -1537.047,E2 -1537.047} C_VEL
LIN {X 0,Y 587.3,Z 375.981,A -85,B 0,C 180,E1 -1538.084,E2 -1538.084} C_VEL
LIN {X 0,Y 587.344,Z 367.526,A -85,B 0,C 180,E1 -1538.95,E2 -1538.95} C_VEL
LIN {X 0,Y 587.415,Z 357.08,A -85,B 0,C 180,E1 -1539.817,E2 -1539.817} C_VEL
LIN {X 0,Y 587.451,Z 346.742,A -85,B 0,C 180,E1 -1540.513,E2 -1540.513} C_VEL
LIN {X 0,Y 587.53,Z 335.153,A -85,B 0,C 180,E1 -1541.134,E2 -1541.134} C_VEL
LIN {X 0,Y 587.595,Z 322.671,A -85,B 0,C 180,E1 -1541.637,E2 -1541.637} C_VEL
LIN {X 0,Y 587.711,Z 309.398,A -85,B 0,C 180,E1 -1542.015,E2 -1542.015} C_VEL
LIN {X 0,Y 587.594,Z 302.103,A -85,B 0,C 180,E1 -1542.162,E2 -1542.162} C_VEL
LIN {X 0,Y 587.193,Z 299.527,A -85,B 0,C 180,E1 -1542.223,E2 -1542.223} C_VEL
LIN {X 0,Y 587.255,Z 289.432,A -85,B 0,C 180,E1 -1544.911,E2 -1544.911} C_VEL
LIN {X 0,Y 587.299,Z 278.841,A -85,B 0,C 180,E1 -1547.768,E2 -1547.768} C_VEL
LIN {X 0,Y 587.379,Z 268.25,A -85,B 0,C 180,E1 -1550.67,E2 -1550.67} C_VEL
LIN {X 0,Y 587.437,Z 257.659,A -85,B 0,C 180,E1 -1553.628,E2 -1553.628} C_VEL
LIN {X 0,Y 587.491,Z 248.391,A -85,B 0,C 180,E1 -1556.272,E2 -1556.272} C_VEL
LIN {X 0,Y 587.492,Z 240.448,A -85,B 0,C 180,E1 -1558.589,E2 -1558.589} C_VEL
LIN {X 0,Y 587.62,Z 231.181,A -85,B 0,C 180,E1 -1561.351,E2 -1561.351} C_VEL
LIN {X 0,Y 587.652,Z 223.237,A -85,B 0,C 180,E1 -1563.788,E2 -1563.788} C_VEL
LIN {X 0,Y 587.629,Z 217.542,A -85,B 0,C 180,E1 -1565.583,E2 -1565.583} C_VEL
LIN {X 0,Y 587.294,Z 215.332,A -85,B 0,C 180,E1 -1566.325,E2 -1566.325} C_VEL
LIN {X 0,Y 587.313,Z 215.329,A -85,B 0,C 180,E1 -1568.939,E2 -1568.939} C_VEL
LIN {X 0,Y 587.335,Z 215.322,A -85,B 0,C 180,E1 -1571.158,E2 -1571.158} C_VEL
LIN {X 0,Y 587.325,Z 215.329,A -85,B 0,C 180,E1 -1574.113,E2 -1574.113} C_VEL
LIN {X 0,Y 587.321,Z 215.323,A -85,B 0,C 180,E1 -1576.994,E2 -1576.994} C_VEL
LIN {X 0,Y 587.313,Z 215.326,A -85,B 0,C 180,E1 -1579.745,E2 -1579.745} C_VEL
LIN {X 0,Y 587.345,Z 215.321,A -85,B 0,C 180,E1 -1582.392,E2 -1582.392} C_VEL
LIN {X 0,Y 587.328,Z 215.321,A -85,B 0,C 180,E1 -1585.656,E2 -1585.656} C_VEL
LIN {X 0,Y 587.338,Z 215.328,A -85,B 0,C 180,E1 -1588.231,E2 -1588.231} C_VEL
LIN {X 0,Y 587.349,Z 215.319,A -85,B 0,C 180,E1 -1590.868,E2 -1590.868} C_VEL
LIN {X 0,Y 587.346,Z 215.323,A -85,B 0,C 180,E1 -1593.823,E2 -1593.823} C_VEL
LIN {X 0,Y 587.325,Z 215.322,A -85,B 0,C 180,E1 -1595.993,E2 -1595.993} C_VEL
LIN {X 0,Y 587.32,Z 215.323,A -85,B 0,C 180,E1 -1598.226,E2 -1598.226} C_VEL
LIN {X 0,Y 587.337,Z 215.322,A -85,B 0,C 180,E1 -1601.151,E2 -1601.151} C_VEL
LIN {X 0,Y 587.297,Z 215.331,A -85,B 0,C 180,E1 -1604.024,E2 -1604.024} C_VEL
LIN {X 0,Y 587.34,Z 215.325,A -85,B 0,C 180,E1 -1606.154,E2 -1606.154} C_VEL
LIN {X 0,Y 587.296,Z 215.326,A -85,B 0,C 180,E1 -1608.962,E2 -1608.962} C_VEL
LIN {X 0,Y 587.331,Z 215.323,A -85,B 0,C 180,E1 -1611.744,E2 -1611.744} C_VEL
LIN {X 0,Y 587.32,Z 215.323,A -85,B 0,C 180,E1 -1613.818,E2 -1613.818} C_VEL
LIN {X 0,Y 587.311,Z 215.324,A -85,B 0,C 180,E1 -1615.883,E2 -1615.883} C_VEL
LIN {X 0,Y 587.368,Z 215.319,A -85,B 0,C 180,E1 -1617.943,E2 -1617.943} C_VEL
LIN {X 0,Y 587.381,Z 215.316,A -85,B 0,C 180,E1 -1620.686,E2 -1620.686} C_VEL
LIN {X 0,Y 587.325,Z 215.326,A -85,B 0,C 180,E1 -1623.43,E2 -1623.43} C_VEL
LIN {X 0,Y 587.345,Z 215.327,A -85,B 0,C 180,E1 -1625.493,E2 -1625.493} C_VEL
LIN {X 0,Y 587.312,Z 215.323,A -85,B 0,C 180,E1 -1628.256,E2 -1628.256} C_VEL
LIN {X 0,Y 587.357,Z 215.321,A -85,B 0,C 180,E1 -1631.134,E2 -1631.134} C_VEL
LIN {X 0,Y 587.364,Z 215.324,A -85,B 0,C 180,E1 -1634.257,E2 -1634.257} C_VEL
LIN {X 0,Y 587.35,Z 215.321,A -85,B 0,C 180,E1 -1637.406,E2 -1637.406} C_VEL
LIN {X 0,Y 587.312,Z 215.326,A -85,B 0,C 180,E1 -1638.259,E2 -1638.259} C_VEL
LIN {X 0,Y 586.67,Z 215.405,A -85,B 0,C 180,E1 -1638.831,E2 -1638.831} C_VEL
LIN {X 0,Y 583.86,Z 215.76,A -85,B 0,C 180,E1 -1639.76,E2 -1639.76} C_VEL
LIN {X 0,Y 581.457,Z 216.056,A -85,B 0,C 180,E1 -1640.507,E2 -1640.507} C_VEL
LIN {X 0,Y 580.395,Z 216.189,A -85,B 0,C 180,E1 -1641.083,E2 -1641.083} C_VEL
LIN {X 0,Y 580.294,Z 216.204,A -85,B 0,C 180,E1 -1641.278,E2 -1641.278} C_VEL
LIN {X 0,Y 580.253,Z 216.206,A -85,B 0,C 180,E1 -1643.559,E2 -1643.559} C_VEL
LIN {X 0,Y 580.252,Z 216.205,A -85,B 0,C 180,E1 -1646.324,E2 -1646.324} C_VEL
LIN {X 0,Y 580.28,Z 216.199,A -85,B 0,C 180,E1 -1649.304,E2 -1649.304} C_VEL
LIN {X 0,Y 580.303,Z 216.203,A -85,B 0,C 180,E1 -1652.201,E2 -1652.201} C_VEL
LIN {X 0,Y 580.294,Z 216.198,A -85,B 0,C 180,E1 -1654.696,E2 -1654.696} C_VEL
LIN {X 0,Y 580.295,Z 216.204,A -85,B 0,C 180,E1 -1657.269,E2 -1657.269} C_VEL
LIN {X 0,Y 580.294,Z 216.198,A -85,B 0,C 180,E1 -1660.27,E2 -1660.27} C_VEL
LIN {X 0,Y 580.278,Z 216.207,A -85,B 0,C 180,E1 -1662.707,E2 -1662.707} C_VEL
LIN {X 0,Y 580.241,Z 216.204,A -85,B 0,C 180,E1 -1665.612,E2 -1665.612} C_VEL
LIN {X 0,Y 580.24,Z 216.209,A -85,B 0,C 180,E1 -1668.227,E2 -1668.227} C_VEL
LIN {X 0,Y 580.271,Z 216.201,A -85,B 0,C 180,E1 -1670.964,E2 -1670.964} C_VEL
LIN {X 0,Y 580.256,Z 216.207,A -85,B 0,C 180,E1 -1673.595,E2 -1673.595} C_VEL
LIN {X 0,Y 580.29,Z 216.198,A -85,B 0,C 180,E1 -1676.143,E2 -1676.143} C_VEL
LIN {X 0,Y 580.221,Z 216.214,A -85,B 0,C 180,E1 -1678.61,E2 -1678.61} C_VEL
LIN {X 0,Y 580.169,Z 216.261,A -85,B 0,C 180,E1 -1679.417,E2 -1679.417} C_VEL
LIN {X 0,Y 580.147,Z 219.448,A -85,B 0,C 180,E1 -1682.17,E2 -1682.17} C_VEL
LIN {X 0,Y 580.128,Z 222.57,A -85,B 0,C 180,E1 -1684.911,E2 -1684.911} C_VEL
LIN {X 0,Y 580.1,Z 225.203,A -85,B 0,C 180,E1 -1687.189,E2 -1687.189} C_VEL
LIN {X 0,Y 580.081,Z 227.793,A -85,B 0,C 180,E1 -1689.429,E2 -1689.429} C_VEL
LIN {X 0,Y 580.037,Z 230.351,A -85,B 0,C 180,E1 -1691.637,E2 -1691.637} C_VEL
LIN {X 0,Y 580.074,Z 233.154,A -85,B 0,C 180,E1 -1693.819,E2 -1693.819} C_VEL
LIN {X 0,Y 580.049,Z 236.918,A -85,B 0,C 180,E1 -1696.69,E2 -1696.69} C_VEL
LIN {X 0,Y 580.046,Z 240.696,A -85,B 0,C 180,E1 -1699.528,E2 -1699.528} C_VEL
LIN {X 0,Y 580.025,Z 243.686,A -85,B 0,C 180,E1 -1701.748,E2 -1701.748} C_VEL
LIN {X 0,Y 580.774,Z 249.631,A -85,B 0,C 180,E1 -1701.89,E2 -1701.89} C_VEL
LIN {X 0,Y 580.688,Z 262.49,A -85,B 0,C 180,E1 -1702.261,E2 -1702.261} C_VEL
LIN {X 0,Y 580.651,Z 273.391,A -85,B 0,C 180,E1 -1702.698,E2 -1702.698} C_VEL
LIN {X 0,Y 580.461,Z 285.266,A -85,B 0,C 180,E1 -1703.313,E2 -1703.313} C_VEL
LIN {X 0,Y 580.434,Z 296.864,A -85,B 0,C 180,E1 -1704.092,E2 -1704.092} C_VEL
LIN {X 0,Y 580.315,Z 307.266,A -85,B 0,C 180,E1 -1704.962,E2 -1704.962} C_VEL
LIN {X 0,Y 580.248,Z 315.722,A -85,B 0,C 180,E1 -1705.832,E2 -1705.832} C_VEL
LIN {X 0,Y 580.197,Z 323.965,A -85,B 0,C 180,E1 -1706.874,E2 -1706.874} C_VEL
LIN {X 0,Y 580.089,Z 330.625,A -85,B 0,C 180,E1 -1707.916,E2 -1707.916} C_VEL
LIN {X 0,Y 580.119,Z 335.948,A -85,B 0,C 180,E1 -1708.958,E2 -1708.958} C_VEL
LIN {X 0,Y 580.066,Z 340.114,A -85,B 0,C 180,E1 -1709.999,E2 -1709.999} C_VEL
LIN {X 0,Y 580.044,Z 342.327,A -85,B 0,C 180,E1 -1710.693,E2 -1710.693} C_VEL
LIN {X 0,Y 580.048,Z 344.071,A -85,B 0,C 180,E1 -1711.388,E2 -1711.388} C_VEL
LIN {X 0,Y 580.039,Z 346.321,A -85,B 0,C 180,E1 -1712.777,E2 -1712.777} C_VEL
LIN {X 0,Y 580.106,Z 346.864,A -85,B 0,C 180,E1 -1713.472,E2 -1713.472} C_VEL
LIN {X 0,Y 580.087,Z 346.979,A -85,B 0,C 180,E1 -1714.168,E2 -1714.168} C_VEL
LIN {X 0,Y 580.09,Z 346.039,A -85,B 0,C 180,E1 -1715.561,E2 -1715.561} C_VEL
LIN {X 0,Y 580.099,Z 344.364,A -85,B 0,C 180,E1 -1716.561,E2 -1716.561} C_VEL
LIN {X 0,Y 580.08,Z 340.408,A -85,B 0,C 180,E1 -1718.008,E2 -1718.008} C_VEL
LIN {X 0,Y 580.072,Z 336.28,A -85,B 0,C 180,E1 -1719.061,E2 -1719.061} C_VEL
LIN {X 0,Y 580.13,Z 329.938,A -85,B 0,C 180,E1 -1720.292,E2 -1720.292} C_VEL
LIN {X 0,Y 580.193,Z 323.008,A -85,B 0,C 180,E1 -1721.351,E2 -1721.351} C_VEL
LIN {X 0,Y 580.263,Z 315.913,A -85,B 0,C 180,E1 -1722.236,E2 -1722.236} C_VEL
LIN {X 0,Y 580.314,Z 307.314,A -85,B 0,C 180,E1 -1723.124,E2 -1723.124} C_VEL
LIN {X 0,Y 580.398,Z 296.663,A -85,B 0,C 180,E1 -1724.014,E2 -1724.014} C_VEL
LIN {X 0,Y 580.482,Z 286.056,A -85,B 0,C 180,E1 -1724.728,E2 -1724.728} C_VEL
LIN {X 0,Y 580.61,Z 274.285,A -85,B 0,C 180,E1 -1725.353,E2 -1725.353} C_VEL
LIN {X 0,Y 580.681,Z 262.001,A -85,B 0,C 180,E1 -1725.846,E2 -1725.846} C_VEL
LIN {X 0,Y 580.771,Z 248.637,A -85,B 0,C 180,E1 -1726.224,E2 -1726.224} C_VEL
LIN {X 0,Y 580.052,Z 243.671,A -85,B 0,C 180,E1 -1726.353,E2 -1726.353} C_VEL
LIN {X 0,Y 580.058,Z 239.984,A -85,B 0,C 180,E1 -1729.094,E2 -1729.094} C_VEL
LIN {X 0,Y 580.046,Z 237.033,A -85,B 0,C 180,E1 -1731.313,E2 -1731.313} C_VEL
LIN {X 0,Y 580.043,Z 234.073,A -85,B 0,C 180,E1 -1733.567,E2 -1733.567} C_VEL
LIN {X 0,Y 580.087,Z 230.546,A -85,B 0,C 180,E1 -1736.292,E2 -1736.292} C_VEL
LIN {X 0,Y 580.119,Z 227.106,A -85,B 0,C 180,E1 -1739.277,E2 -1739.277} C_VEL
LIN {X 0,Y 580.122,Z 223.783,A -85,B 0,C 180,E1 -1742.21,E2 -1742.21} C_VEL
LIN {X 0,Y 580.136,Z 220.884,A -85,B 0,C 180,E1 -1744.705,E2 -1744.705} C_VEL
LIN {X 0,Y 580.152,Z 217.919,A -85,B 0,C 180,E1 -1747.278,E2 -1747.278} C_VEL
LIN {X 0,Y 580.203,Z 216.217,A -85,B 0,C 180,E1 -1749.039,E2 -1749.039} C_VEL
LIN {X 0,Y 580.31,Z 216.197,A -85,B 0,C 180,E1 -1751.764,E2 -1751.764} C_VEL
LIN {X 0,Y 580.261,Z 216.206,A -85,B 0,C 180,E1 -1754.625,E2 -1754.625} C_VEL
LIN {X 0,Y 580.277,Z 216.208,A -85,B 0,C 180,E1 -1757.627,E2 -1757.627} C_VEL
LIN {X 0,Y 580.276,Z 216.201,A -85,B 0,C 180,E1 -1760.065,E2 -1760.065} C_VEL
LIN {X 0,Y 580.295,Z 216.199,A -85,B 0,C 180,E1 -1763.064,E2 -1763.064} C_VEL
LIN {X 0,Y 580.292,Z 216.2,A -85,B 0,C 180,E1 -1765.44,E2 -1765.44} C_VEL
LIN {X 0,Y 580.292,Z 216.2,A -85,B 0,C 180,E1 -1767.969,E2 -1767.969} C_VEL
LIN {X 0,Y 580.284,Z 216.204,A -85,B 0,C 180,E1 -1771.023,E2 -1771.023} C_VEL
LIN {X 0,Y 580.32,Z 216.196,A -85,B 0,C 180,E1 -1773.657,E2 -1773.657} C_VEL
LIN {X 0,Y 580.27,Z 216.202,A -85,B 0,C 180,E1 -1776.441,E2 -1776.441} C_VEL
LIN {X 0,Y 580.257,Z 216.205,A -85,B 0,C 180,E1 -1779.436,E2 -1779.436} C_VEL
LIN {X 0,Y 580.251,Z 216.204,A -85,B 0,C 180,E1 -1781.644,E2 -1781.644} C_VEL
LIN {X 0,Y 580.274,Z 216.205,A -85,B 0,C 180,E1 -1783.825,E2 -1783.825} C_VEL
LIN {X 0,Y 580.317,Z 216.198,A -85,B 0,C 180,E1 -1785.983,E2 -1785.983} C_VEL
LIN {X 0,Y 580.341,Z 216.198,A -85,B 0,C 180,E1 -1788.827,E2 -1788.827} C_VEL
LIN {X 0,Y 580.321,Z 216.201,A -85,B 0,C 180,E1 -1792.344,E2 -1792.344} C_VEL
LIN {X 0,Y 580.337,Z 216.195,A -85,B 0,C 180,E1 -1795.137,E2 -1795.137} C_VEL
LIN {X 0,Y 580.318,Z 216.195,A -85,B 0,C 180,E1 -1797.918,E2 -1797.918} C_VEL
LIN {X 0,Y 580.349,Z 216.196,A -85,B 0,C 180,E1 -1800.694,E2 -1800.694} C_VEL
LIN {X 0,Y 580.27,Z 216.204,A -85,B 0,C 180,E1 -1803.472,E2 -1803.472} C_VEL
LIN {X 0,Y 580.32,Z 216.2,A -85,B 0,C 180,E1 -1805.56,E2 -1805.56} C_VEL
LIN {X 0,Y 580.323,Z 216.197,A -85,B 0,C 180,E1 -1808.356,E2 -1808.356} C_VEL
LIN {X 0,Y 580.288,Z 216.199,A -85,B 0,C 180,E1 -1811.191,E2 -1811.191} C_VEL
LIN {X 0,Y 580.314,Z 216.198,A -85,B 0,C 180,E1 -1814.017,E2 -1814.017} C_VEL
LIN {X 0,Y 580.302,Z 216.204,A -85,B 0,C 180,E1 -1816.915,E2 -1816.915} C_VEL
LIN {X 0,Y 580.292,Z 216.2,A -85,B 0,C 180,E1 -1819.823,E2 -1819.823} C_VEL
LIN {X 0,Y 580.239,Z 216.21,A -85,B 0,C 180,E1 -1822.054,E2 -1822.054} C_VEL
LIN {X 0,Y 580.3,Z 216.203,A -85,B 0,C 180,E1 -1825.08,E2 -1825.08} C_VEL
LIN {X 0,Y 580.312,Z 216.197,A -85,B 0,C 180,E1 -1827.864,E2 -1827.864} C_VEL
LIN {X 0,Y 580.279,Z 216.201,A -85,B 0,C 180,E1 -1830.696,E2 -1830.696} C_VEL
LIN {X 0,Y 580.292,Z 216.204,A -85,B 0,C 180,E1 -1833.317,E2 -1833.317} C_VEL
LIN {X 0,Y 580.238,Z 216.206,A -85,B 0,C 180,E1 -1835.757,E2 -1835.757} C_VEL
LIN {X 0,Y 580.282,Z 216.204,A -85,B 0,C 180,E1 -1838.147,E2 -1838.147} C_VEL
LIN {X 0,Y 580.292,Z 216.199,A -85,B 0,C 180,E1 -1840.844,E2 -1840.844} C_VEL
LIN {X 0,Y 580.26,Z 216.205,A -85,B 0,C 180,E1 -1843.66,E2 -1843.66} C_VEL
LIN {X 0,Y 580.271,Z 216.208,A -85,B 0,C 180,E1 -1846.61,E2 -1846.61} C_VEL
LIN {X 0,Y 580.3,Z 216.199,A -85,B 0,C 180,E1 -1849.158,E2 -1849.158} C_VEL
LIN {X 0,Y 580.283,Z 216.205,A -85,B 0,C 180,E1 -1851.928,E2 -1851.928} C_VEL
LIN {X 0,Y 580.309,Z 216.334,A -85,B 0,C 180,E1 -1853.506,E2 -1853.506} C_VEL
LIN {X 0,Y 580.731,Z 220.597,A -85,B 0,C 180,E1 -1854.913,E2 -1854.913} C_VEL
LIN {X 0,Y 580.69,Z 229.865,A -85,B 0,C 180,E1 -1857.825,E2 -1857.825} C_VEL
LIN {X 0,Y 580.564,Z 239.138,A -85,B 0,C 180,E1 -1860.645,E2 -1860.645} C_VEL
LIN {X 0,Y 580.475,Z 248.399,A -85,B 0,C 180,E1 -1863.388,E2 -1863.388} C_VEL
LIN {X 0,Y 580.421,Z 257.666,A -85,B 0,C 180,E1 -1866.071,E2 -1866.071} C_VEL
LIN {X 0,Y 580.319,Z 267.409,A -85,B 0,C 180,E1 -1868.831,E2 -1868.831} C_VEL
LIN {X 0,Y 580.258,Z 276.201,A -85,B 0,C 180,E1 -1871.28,E2 -1871.28} C_VEL
LIN {X 0,Y 580.211,Z 285.468,A -85,B 0,C 180,E1 -1873.825,E2 -1873.825} C_VEL
LIN {X 0,Y 580.184,Z 296.059,A -85,B 0,C 180,E1 -1876.695,E2 -1876.695} C_VEL
LIN {X 0,Y 580.118,Z 299.534,A -85,B 0,C 180,E1 -1877.628,E2 -1877.628} C_VEL
LIN {X 0,Y 580.798,Z 305.288,A -85,B 0,C 180,E1 -1877.753,E2 -1877.753} C_VEL
LIN {X 0,Y 580.732,Z 318.535,A -85,B 0,C 180,E1 -1878.084,E2 -1878.084} C_VEL
LIN {X 0,Y 580.615,Z 330.346,A -85,B 0,C 180,E1 -1878.516,E2 -1878.516} C_VEL
LIN {X 0,Y 580.506,Z 342.229,A -85,B 0,C 180,E1 -1879.097,E2 -1879.097} C_VEL
LIN {X 0,Y 580.446,Z 353.493,A -85,B 0,C 180,E1 -1879.801,E2 -1879.801} C_VEL
LIN {X 0,Y 580.352,Z 363.659,A -85,B 0,C 180,E1 -1880.592,E2 -1880.592} C_VEL
LIN {X 0,Y 580.279,Z 372.797,A -85,B 0,C 180,E1 -1881.469,E2 -1881.469} C_VEL
LIN {X 0,Y 580.198,Z 381.699,A -85,B 0,C 180,E1 -1882.519,E2 -1882.519} C_VEL
LIN {X 0,Y 580.119,Z 388.468,A -85,B 0,C 180,E1 -1883.505,E2 -1883.505} C_VEL
LIN {X 0,Y 580.139,Z 393.686,A -85,B 0,C 180,E1 -1884.44,E2 -1884.44} C_VEL
LIN {X 0,Y 580.108,Z 398.376,A -85,B 0,C 180,E1 -1885.484,E2 -1885.484} C_VEL
LIN {X 0,Y 580.122,Z 401.959,A -85,B 0,C 180,E1 -1886.528,E2 -1886.528} C_VEL
LIN {X 0,Y 580.043,Z 403.811,A -85,B 0,C 180,E1 -1887.223,E2 -1887.223} C_VEL
LIN {X 0,Y 580.04,Z 405.203,A -85,B 0,C 180,E1 -1887.918,E2 -1887.918} C_VEL
LIN {X 0,Y 580.04,Z 406.785,A -85,B 0,C 180,E1 -1889.307,E2 -1889.307} C_VEL
LIN {X 0,Y 580.037,Z 407,A -85,B 0,C 180,E1 -1890.001,E2 -1890.001} C_VEL
LIN {X 0,Y 580.047,Z 406.184,A -85,B 0,C 180,E1 -1891.39,E2 -1891.39} C_VEL
LIN {X 0,Y 580.04,Z 405.2,A -85,B 0,C 180,E1 -1892.084,E2 -1892.084} C_VEL
LIN {X 0,Y 580.043,Z 403.807,A -85,B 0,C 180,E1 -1892.779,E2 -1892.779} C_VEL
LIN {X 0,Y 580.11,Z 400.893,A -85,B 0,C 180,E1 -1893.822,E2 -1893.822} C_VEL
LIN {X 0,Y 580.053,Z 396.946,A -85,B 0,C 180,E1 -1894.866,E2 -1894.866} C_VEL
LIN {X 0,Y 580.139,Z 390.872,A -85,B 0,C 180,E1 -1896.086,E2 -1896.086} C_VEL
LIN {X 0,Y 580.185,Z 384.229,A -85,B 0,C 180,E1 -1897.133,E2 -1897.133} C_VEL
LIN {X 0,Y 580.251,Z 375.981,A -85,B 0,C 180,E1 -1898.183,E2 -1898.183} C_VEL
LIN {X 0,Y 580.308,Z 367.527,A -85,B 0,C 180,E1 -1899.059,E2 -1899.059} C_VEL
LIN {X 0,Y 580.412,Z 357.081,A -85,B 0,C 180,E1 -1899.937,E2 -1899.937} C_VEL
LIN {X 0,Y 580.454,Z 346.743,A -85,B 0,C 180,E1 -1900.641,E2 -1900.641} C_VEL
LIN {X 0,Y 580.565,Z 335.574,A -85,B 0,C 180,E1 -1901.248,E2 -1901.248} C_VEL
LIN {X 0,Y 580.629,Z 323.739,A -85,B 0,C 180,E1 -1901.743,E2 -1901.743} C_VEL
LIN {X 0,Y 580.769,Z 310.312,A -85,B 0,C 180,E1 -1902.138,E2 -1902.138} C_VEL
LIN {X 0,Y 580.589,Z 302.438,A -85,B 0,C 180,E1 -1902.306,E2 -1902.306} C_VEL
LIN {X 0,Y 580.119,Z 299.527,A -85,B 0,C 180,E1 -1902.374,E2 -1902.374} C_VEL
LIN {X 0,Y 580.217,Z 289.432,A -85,B 0,C 180,E1 -1905.096,E2 -1905.096} C_VEL
LIN {X 0,Y 580.249,Z 278.841,A -85,B 0,C 180,E1 -1907.991,E2 -1907.991} C_VEL
LIN {X 0,Y 580.347,Z 268.488,A -85,B 0,C 180,E1 -1910.865,E2 -1910.865} C_VEL
LIN {X 0,Y 580.409,Z 258.983,A -85,B 0,C 180,E1 -1913.553,E2 -1913.553} C_VEL
LIN {X 0,Y 580.487,Z 249.217,A -85,B 0,C 180,E1 -1916.372,E2 -1916.372} C_VEL
LIN {X 0,Y 580.517,Z 240.448,A -85,B 0,C 180,E1 -1918.965,E2 -1918.965} C_VEL
LIN {X 0,Y 580.658,Z 231.328,A -85,B 0,C 180,E1 -1921.725,E2 -1921.725} C_VEL
LIN {X 0,Y 580.714,Z 223.317,A -85,B 0,C 180,E1 -1924.223,E2 -1924.223} C_VEL
LIN {X 0,Y 580.63,Z 218.376,A -85,B 0,C 180,E1 -1925.809,E2 -1925.809} C_VEL
LIN {X 0,Y 580.277,Z 216.207,A -85,B 0,C 180,E1 -1926.593,E2 -1926.593} C_VEL
LIN {X 0,Y 580.289,Z 216.201,A -85,B 0,C 180,E1 -1929.184,E2 -1929.184} C_VEL
LIN {X 0,Y 580.282,Z 216.202,A -85,B 0,C 180,E1 -1931.77,E2 -1931.77} C_VEL
LIN {X 0,Y 580.272,Z 216.202,A -85,B 0,C 180,E1 -1934.627,E2 -1934.627} C_VEL
LIN {X 0,Y 580.293,Z 216.206,A -85,B 0,C 180,E1 -1937.629,E2 -1937.629} C_VEL
LIN {X 0,Y 580.287,Z 216.199,A -85,B 0,C 180,E1 -1940.067,E2 -1940.067} C_VEL
LIN {X 0,Y 580.282,Z 216.204,A -85,B 0,C 180,E1 -1943.069,E2 -1943.069} C_VEL
LIN {X 0,Y 580.271,Z 216.204,A -85,B 0,C 180,E1 -1946.142,E2 -1946.142} C_VEL
LIN {X 0,Y 580.271,Z 216.203,A -85,B 0,C 180,E1 -1948.614,E2 -1948.614} C_VEL
LIN {X 0,Y 580.291,Z 216.198,A -85,B 0,C 180,E1 -1951.024,E2 -1951.024} C_VEL
LIN {X 0,Y 580.286,Z 216.2,A -85,B 0,C 180,E1 -1954.151,E2 -1954.151} C_VEL
LIN {X 0,Y 580.275,Z 216.201,A -85,B 0,C 180,E1 -1956.442,E2 -1956.442} C_VEL
LIN {X 0,Y 580.274,Z 216.201,A -85,B 0,C 180,E1 -1959.437,E2 -1959.437} C_VEL
LIN {X 0,Y 580.252,Z 216.203,A -85,B 0,C 180,E1 -1961.645,E2 -1961.645} C_VEL
LIN {X 0,Y 580.272,Z 216.203,A -85,B 0,C 180,E1 -1964.547,E2 -1964.547} C_VEL
LIN {X 0,Y 580.238,Z 216.204,A -85,B 0,C 180,E1 -1966.695,E2 -1966.695} C_VEL
LIN {X 0,Y 580.274,Z 216.2,A -85,B 0,C 180,E1 -1968.826,E2 -1968.826} C_VEL
LIN {X 0,Y 580.303,Z 216.2,A -85,B 0,C 180,E1 -1971.644,E2 -1971.644} C_VEL
LIN {X 0,Y 580.28,Z 216.2,A -85,B 0,C 180,E1 -1973.742,E2 -1973.742} C_VEL
LIN {X 0,Y 580.267,Z 216.201,A -85,B 0,C 180,E1 -1975.833,E2 -1975.833} C_VEL
LIN {X 0,Y 580.34,Z 216.194,A -85,B 0,C 180,E1 -1977.918,E2 -1977.918} C_VEL
LIN {X 0,Y 580.353,Z 216.192,A -85,B 0,C 180,E1 -1980.694,E2 -1980.694} C_VEL
LIN {X 0,Y 580.276,Z 216.205,A -85,B 0,C 180,E1 -1983.472,E2 -1983.472} C_VEL
LIN {X 0,Y 580.309,Z 216.202,A -85,B 0,C 180,E1 -1985.56,E2 -1985.56} C_VEL
LIN {X 0,Y 580.288,Z 216.198,A -85,B 0,C 180,E1 -1988.357,E2 -1988.357} C_VEL
LIN {X 0,Y 580.308,Z 216.198,A -85,B 0,C 180,E1 -1991.191,E2 -1991.191} C_VEL
LIN {X 0,Y 580.322,Z 216.198,A -85,B 0,C 180,E1 -1994.017,E2 -1994.017} C_VEL
LIN {X 0,Y 580.321,Z 216.195,A -85,B 0,C 180,E1 -1996.914,E2 -1996.914} C_VEL
LIN {X 0,Y 580.289,Z 216.204,A -85,B 0,C 180,E1 -1999.823,E2 -1999.823} C_VEL
LIN {X 0,Y 580.294,Z 216.204,A -85,B 0,C 180,E1 -2001.278,E2 -2001.278} C_VEL
LIN {X 0,Y 579.579,Z 216.298,A -85,B 0,C 180,E1 -2001.857,E2 -2001.857} C_VEL
LIN {X 0,Y 576.691,Z 216.655,A -85,B 0,C 180,E1 -2002.797,E2 -2002.797} C_VEL
LIN {X 0,Y 574.286,Z 216.949,A -85,B 0,C 180,E1 -2003.553,E2 -2003.553} C_VEL
LIN {X 0,Y 573.269,Z 217.073,A -85,B 0,C 180,E1 -2004.137,E2 -2004.137} C_VEL
LIN {X 0,Y 573.193,Z 217.083,A -85,B 0,C 180,E1 -2004.335,E2 -2004.335} C_VEL
LIN {X 0,Y 573.187,Z 217.087,A -85,B 0,C 180,E1 -2006.979,E2 -2006.979} C_VEL
LIN {X 0,Y 573.226,Z 217.078,A -85,B 0,C 180,E1 -2009.483,E2 -2009.483} C_VEL
LIN {X 0,Y 573.256,Z 217.08,A -85,B 0,C 180,E1 -2012.227,E2 -2012.227} C_VEL
LIN {X 0,Y 573.213,Z 217.082,A -85,B 0,C 180,E1 -2015.188,E2 -2015.188} C_VEL
LIN {X 0,Y 573.237,Z 217.08,A -85,B 0,C 180,E1 -2017.808,E2 -2017.808} C_VEL
LIN {X 0,Y 573.253,Z 217.077,A -85,B 0,C 180,E1 -2020.525,E2 -2020.525} C_VEL
LIN {X 0,Y 573.214,Z 217.08,A -85,B 0,C 180,E1 -2023.362,E2 -2023.362} C_VEL
LIN {X 0,Y 573.199,Z 217.088,A -85,B 0,C 180,E1 -2026.336,E2 -2026.336} C_VEL
LIN {X 0,Y 573.195,Z 217.083,A -85,B 0,C 180,E1 -2028.539,E2 -2028.539} C_VEL
LIN {X 0,Y 573.24,Z 217.08,A -85,B 0,C 180,E1 -2031.297,E2 -2031.297} C_VEL
LIN {X 0,Y 573.201,Z 217.082,A -85,B 0,C 180,E1 -2034.021,E2 -2034.021} C_VEL
LIN {X 0,Y 573.24,Z 217.079,A -85,B 0,C 180,E1 -2036.515,E2 -2036.515} C_VEL
LIN {X 0,Y 573.15,Z 217.095,A -85,B 0,C 180,E1 -2039.132,E2 -2039.132} C_VEL
LIN {X 0,Y 573.101,Z 217.398,A -85,B 0,C 180,E1 -2039.814,E2 -2039.814} C_VEL
LIN {X 0,Y 573.096,Z 220.168,A -85,B 0,C 180,E1 -2042.224,E2 -2042.224} C_VEL
LIN {X 0,Y 573.087,Z 223.512,A -85,B 0,C 180,E1 -2045.162,E2 -2045.162} C_VEL
LIN {X 0,Y 573.005,Z 226.358,A -85,B 0,C 180,E1 -2047.652,E2 -2047.652} C_VEL
LIN {X 0,Y 572.978,Z 228.947,A -85,B 0,C 180,E1 -2049.912,E2 -2049.912} C_VEL
LIN {X 0,Y 572.976,Z 232.352,A -85,B 0,C 180,E1 -2052.879,E2 -2052.879} C_VEL
LIN {X 0,Y 572.98,Z 236.046,A -85,B 0,C 180,E1 -2055.799,E2 -2055.799} C_VEL
LIN {X 0,Y 572.986,Z 240.092,A -85,B 0,C 180,E1 -2058.888,E2 -2058.888} C_VEL
LIN {X 0,Y 572.962,Z 243.666,A -85,B 0,C 180,E1 -2061.579,E2 -2061.579} C_VEL
LIN {X 0,Y 573.849,Z 250.782,A -85,B 0,C 180,E1 -2061.77,E2 -2061.77} C_VEL
LIN {X 0,Y 573.747,Z 263.947,A -85,B 0,C 180,E1 -2062.167,E2 -2062.167} C_VEL
LIN {X 0,Y 573.641,Z 276.307,A -85,B 0,C 180,E1 -2062.696,E2 -2062.696} C_VEL
LIN {X 0,Y 573.476,Z 287.878,A -85,B 0,C 180,E1 -2063.344,E2 -2063.344} C_VEL
LIN {X 0,Y 573.404,Z 298.674,A -85,B 0,C 180,E1 -2064.107,E2 -2064.107} C_VEL
LIN {X 0,Y 573.273,Z 307.803,A -85,B 0,C 180,E1 -2064.9,E2 -2064.9} C_VEL
LIN {X 0,Y 573.202,Z 316.145,A -85,B 0,C 180,E1 -2065.78,E2 -2065.78} C_VEL
LIN {X 0,Y 573.139,Z 324.316,A -85,B 0,C 180,E1 -2066.836,E2 -2066.836} C_VEL
LIN {X 0,Y 573.001,Z 330.912,A -85,B 0,C 180,E1 -2067.89,E2 -2067.89} C_VEL
LIN {X 0,Y 573.039,Z 336.177,A -85,B 0,C 180,E1 -2068.945,E2 -2068.945} C_VEL
LIN {X 0,Y 572.969,Z 340.29,A -85,B 0,C 180,E1 -2069.999,E2 -2069.999} C_VEL
LIN {X 0,Y 572.946,Z 342.469,A -85,B 0,C 180,E1 -2070.702,E2 -2070.702} C_VEL
LIN {X 0,Y 572.947,Z 344.173,A -85,B 0,C 180,E1 -2071.405,E2 -2071.405} C_VEL
LIN {X 0,Y 572.954,Z 346.377,A -85,B 0,C 180,E1 -2072.811,E2 -2072.811} C_VEL
LIN {X 0,Y 573.006,Z 346.886,A -85,B 0,C 180,E1 -2073.515,E2 -2073.515} C_VEL
LIN {X 0,Y 573.007,Z 346.968,A -85,B 0,C 180,E1 -2074.219,E2 -2074.219} C_VEL
LIN {X 0,Y 572.992,Z 345.981,A -85,B 0,C 180,E1 -2075.63,E2 -2075.63} C_VEL
LIN {X 0,Y 573.009,Z 344.455,A -85,B 0,C 180,E1 -2076.548,E2 -2076.548} C_VEL
LIN {X 0,Y 572.993,Z 341.38,A -85,B 0,C 180,E1 -2077.753,E2 -2077.753} C_VEL
LIN {X 0,Y 573.006,Z 337.565,A -85,B 0,C 180,E1 -2078.818,E2 -2078.818} C_VEL
LIN {X 0,Y 573.042,Z 332.603,A -85,B 0,C 180,E1 -2079.886,E2 -2079.886} C_VEL
LIN {X 0,Y 573.13,Z 326.772,A -85,B 0,C 180,E1 -2080.888,E2 -2080.888} C_VEL
LIN {X 0,Y 573.163,Z 319.918,A -85,B 0,C 180,E1 -2081.851,E2 -2081.851} C_VEL
LIN {X 0,Y 573.239,Z 312.189,A -85,B 0,C 180,E1 -2082.748,E2 -2082.748} C_VEL
LIN {X 0,Y 573.346,Z 302.743,A -85,B 0,C 180,E1 -2083.647,E2 -2083.647} C_VEL
LIN {X 0,Y 573.436,Z 291.88,A -85,B 0,C 180,E1 -2084.482,E2 -2084.482} C_VEL
LIN {X 0,Y 573.552,Z 280.445,A -85,B 0,C 180,E1 -2085.183,E2 -2085.183} C_VEL
LIN {X 0,Y 573.707,Z 267.89,A -85,B 0,C 180,E1 -2085.77,E2 -2085.77} C_VEL
LIN {X 0,Y 573.822,Z 254.568,A -85,B 0,C 180,E1 -2086.223,E2 -2086.223} C_VEL
LIN {X 0,Y 573.61,Z 247.8,A -85,B 0,C 180,E1 -2086.398,E2 -2086.398} C_VEL
LIN {X 0,Y 572.989,Z 243.667,A -85,B 0,C 180,E1 -2086.51,E2 -2086.51} C_VEL
LIN {X 0,Y 572.948,Z 239.911,A -85,B 0,C 180,E1 -2089.34,E2 -2089.34} C_VEL
LIN {X 0,Y 572.939,Z 236.959,A -85,B 0,C 180,E1 -2091.591,E2 -2091.591} C_VEL
LIN {X 0,Y 572.976,Z 233.998,A -85,B 0,C 180,E1 -2093.875,E2 -2093.875} C_VEL
LIN {X 0,Y 573.024,Z 230.961,A -85,B 0,C 180,E1 -2096.449,E2 -2096.449} C_VEL
LIN {X 0,Y 573.066,Z 227.51,A -85,B 0,C 180,E1 -2099.455,E2 -2099.455} C_VEL
LIN {X 0,Y 573.059,Z 224.383,A -85,B 0,C 180,E1 -2102.197,E2 -2102.197} C_VEL
LIN {X 0,Y 573.072,Z 220.97,A -85,B 0,C 180,E1 -2105.196,E2 -2105.196} C_VEL
LIN {X 0,Y 573.114,Z 217.986,A -85,B 0,C 180,E1 -2107.815,E2 -2107.815} C_VEL
LIN {X 0,Y 573.103,Z 217.101,A -85,B 0,C 180,E1 -2108.711,E2 -2108.711} C_VEL
LIN {X 0,Y 573.239,Z 217.078,A -85,B 0,C 180,E1 -2110.524,E2 -2110.524} C_VEL
LIN {X 0,Y 573.234,Z 217.078,A -85,B 0,C 180,E1 -2113.358,E2 -2113.358} C_VEL
LIN {X 0,Y 573.227,Z 217.082,A -85,B 0,C 180,E1 -2116.331,E2 -2116.331} C_VEL
LIN {X 0,Y 573.216,Z 217.08,A -85,B 0,C 180,E1 -2118.541,E2 -2118.541} C_VEL
LIN {X 0,Y 573.237,Z 217.08,A -85,B 0,C 180,E1 -2121.298,E2 -2121.298} C_VEL
LIN {X 0,Y 573.257,Z 217.079,A -85,B 0,C 180,E1 -2124.01,E2 -2124.01} C_VEL
LIN {X 0,Y 573.23,Z 217.079,A -85,B 0,C 180,E1 -2126.515,E2 -2126.515} C_VEL
LIN {X 0,Y 573.211,Z 217.087,A -85,B 0,C 180,E1 -2129.118,E2 -2129.118} C_VEL
LIN {X 0,Y 573.255,Z 217.076,A -85,B 0,C 180,E1 -2131.968,E2 -2131.968} C_VEL
LIN {X 0,Y 573.249,Z 217.077,A -85,B 0,C 180,E1 -2134.589,E2 -2134.589} C_VEL
LIN {X 0,Y 573.221,Z 217.083,A -85,B 0,C 180,E1 -2137.661,E2 -2137.661} C_VEL
LIN {X 0,Y 573.254,Z 217.082,A -85,B 0,C 180,E1 -2140.669,E2 -2140.669} C_VEL
LIN {X 0,Y 573.245,Z 217.079,A -85,B 0,C 180,E1 -2143.621,E2 -2143.621} C_VEL
LIN {X 0,Y 573.263,Z 217.079,A -85,B 0,C 180,E1 -2145.807,E2 -2145.807} C_VEL
LIN {X 0,Y 573.272,Z 217.077,A -85,B 0,C 180,E1 -2148.734,E2 -2148.734} C_VEL
LIN {X 0,Y 573.27,Z 217.074,A -85,B 0,C 180,E1 -2151.54,E2 -2151.54} C_VEL
LIN {X 0,Y 573.297,Z 217.071,A -85,B 0,C 180,E1 -2154.372,E2 -2154.372} C_VEL
LIN {X 0,Y 573.299,Z 217.077,A -85,B 0,C 180,E1 -2157.189,E2 -2157.189} C_VEL
LIN {X 0,Y 573.295,Z 217.072,A -85,B 0,C 180,E1 -2160,E2 -2160} C_VEL
LIN {X 0,Y 573.296,Z 217.07,A -85,B 0,C 180,E1 -2162.811,E2 -2162.811} C_VEL
LIN {X 0,Y 573.286,Z 217.076,A -85,B 0,C 180,E1 -2165.628,E2 -2165.628} C_VEL
LIN {X 0,Y 573.278,Z 217.076,A -85,B 0,C 180,E1 -2168.46,E2 -2168.46} C_VEL
LIN {X 0,Y 573.259,Z 217.075,A -85,B 0,C 180,E1 -2171.312,E2 -2171.312} C_VEL
LIN {X 0,Y 573.27,Z 217.073,A -85,B 0,C 180,E1 -2174.425,E2 -2174.425} C_VEL
LIN {X 0,Y 573.25,Z 217.081,A -85,B 0,C 180,E1 -2177.112,E2 -2177.112} C_VEL
LIN {X 0,Y 573.239,Z 217.081,A -85,B 0,C 180,E1 -2180.077,E2 -2180.077} C_VEL
LIN {X 0,Y 573.223,Z 217.081,A -85,B 0,C 180,E1 -2183.1,E2 -2183.1} C_VEL
LIN {X 0,Y 573.249,Z 217.08,A -85,B 0,C 180,E1 -2185.41,E2 -2185.41} C_VEL
LIN {X 0,Y 573.256,Z 217.077,A -85,B 0,C 180,E1 -2188.033,E2 -2188.033} C_VEL
LIN {X 0,Y 573.221,Z 217.08,A -85,B 0,C 180,E1 -2190.883,E2 -2190.883} C_VEL
LIN {X 0,Y 573.253,Z 217.082,A -85,B 0,C 180,E1 -2193.525,E2 -2193.525} C_VEL
LIN {X 0,Y 573.206,Z 217.082,A -85,B 0,C 180,E1 -2196.052,E2 -2196.052} C_VEL
LIN {X 0,Y 573.241,Z 217.08,A -85,B 0,C 180,E1 -2198.702,E2 -2198.702} C_VEL
LIN {X 0,Y 573.218,Z 217.084,A -85,B 0,C 180,E1 -2201.458,E2 -2201.458} C_VEL
LIN {X 0,Y 573.216,Z 217.081,A -85,B 0,C 180,E1 -2204.335,E2 -2204.335} C_VEL
LIN {X 0,Y 573.234,Z 217.079,A -85,B 0,C 180,E1 -2207.359,E2 -2207.359} C_VEL
LIN {X 0,Y 573.244,Z 217.08,A -85,B 0,C 180,E1 -2210.394,E2 -2210.394} C_VEL
LIN {X 0,Y 573.267,Z 217.123,A -85,B 0,C 180,E1 -2213.245,E2 -2213.245} C_VEL
LIN {X 0,Y 573.784,Z 221.921,A -85,B 0,C 180,E1 -2214.854,E2 -2214.854} C_VEL
LIN {X 0,Y 573.696,Z 229.865,A -85,B 0,C 180,E1 -2217.385,E2 -2217.385} C_VEL
LIN {X 0,Y 573.6,Z 237.808,A -85,B 0,C 180,E1 -2219.846,E2 -2219.846} C_VEL
LIN {X 0,Y 573.504,Z 247.075,A -85,B 0,C 180,E1 -2222.644,E2 -2222.644} C_VEL
LIN {X 0,Y 573.429,Z 256.342,A -85,B 0,C 180,E1 -2225.374,E2 -2225.374} C_VEL
LIN {X 0,Y 573.323,Z 266.934,A -85,B 0,C 180,E1 -2228.424,E2 -2228.424} C_VEL
LIN {X 0,Y 573.217,Z 276.334,A -85,B 0,C 180,E1 -2231.079,E2 -2231.079} C_VEL
LIN {X 0,Y 573.157,Z 286.792,A -85,B 0,C 180,E1 -2233.986,E2 -2233.986} C_VEL
LIN {X 0,Y 573.096,Z 297.383,A -85,B 0,C 180,E1 -2236.888,E2 -2236.888} C_VEL
LIN {X 0,Y 573.077,Z 299.534,A -85,B 0,C 180,E1 -2237.473,E2 -2237.473} C_VEL
LIN {X 0,Y 573.869,Z 305.288,A -85,B 0,C 180,E1 -2237.603,E2 -2237.603} C_VEL
LIN {X 0,Y 573.773,Z 318.535,A -85,B 0,C 180,E1 -2237.938,E2 -2237.938} C_VEL
LIN {X 0,Y 573.648,Z 330.876,A -85,B 0,C 180,E1 -2238.398,E2 -2238.398} C_VEL
LIN {X 0,Y 573.523,Z 342.63,A -85,B 0,C 180,E1 -2238.985,E2 -2238.985} C_VEL
LIN {X 0,Y 573.441,Z 353.494,A -85,B 0,C 180,E1 -2239.676,E2 -2239.676} C_VEL
LIN {X 0,Y 573.307,Z 363.659,A -85,B 0,C 180,E1 -2240.475,E2 -2240.475} C_VEL
LIN {X 0,Y 573.214,Z 372.797,A -85,B 0,C 180,E1 -2241.363,E2 -2241.363} C_VEL
LIN {X 0,Y 573.141,Z 381.699,A -85,B 0,C 180,E1 -2242.426,E2 -2242.426} C_VEL
LIN {X 0,Y 573.05,Z 388.409,A -85,B 0,C 180,E1 -2243.415,E2 -2243.415} C_VEL
LIN {X 0,Y 573.07,Z 393.686,A -85,B 0,C 180,E1 -2244.371,E2 -2244.371} C_VEL
LIN {X 0,Y 573.028,Z 398.376,A -85,B 0,C 180,E1 -2245.429,E2 -2245.429} C_VEL
LIN {X 0,Y 573.022,Z 401.96,A -85,B 0,C 180,E1 -2246.485,E2 -2246.485} C_VEL
LIN {X 0,Y 572.959,Z 403.811,A -85,B 0,C 180,E1 -2247.189,E2 -2247.189} C_VEL
LIN {X 0,Y 572.94,Z 405.202,A -85,B 0,C 180,E1 -2247.892,E2 -2247.892} C_VEL
LIN {X 0,Y 572.941,Z 406.785,A -85,B 0,C 180,E1 -2249.298,E2 -2249.298} C_VEL
LIN {X 0,Y 572.938,Z 407,A -85,B 0,C 180,E1 -2250.001,E2 -2250.001} C_VEL
LIN {X 0,Y 572.946,Z 406.184,A -85,B 0,C 180,E1 -2251.407,E2 -2251.407} C_VEL
LIN {X 0,Y 572.94,Z 405.2,A -85,B 0,C 180,E1 -2252.11,E2 -2252.11} C_VEL
LIN {X 0,Y 572.959,Z 403.807,A -85,B 0,C 180,E1 -2252.813,E2 -2252.813} C_VEL
LIN {X 0,Y 573.015,Z 400.893,A -85,B 0,C 180,E1 -2253.869,E2 -2253.869} C_VEL
LIN {X 0,Y 572.963,Z 396.945,A -85,B 0,C 180,E1 -2254.927,E2 -2254.927} C_VEL
LIN {X 0,Y 573.065,Z 390.872,A -85,B 0,C 180,E1 -2256.161,E2 -2256.161} C_VEL
LIN {X 0,Y 573.12,Z 384.229,A -85,B 0,C 180,E1 -2257.222,E2 -2257.222} C_VEL
LIN {X 0,Y 573.199,Z 375.982,A -85,B 0,C 180,E1 -2258.284,E2 -2258.284} C_VEL
LIN {X 0,Y 573.287,Z 367.527,A -85,B 0,C 180,E1 -2259.171,E2 -2259.171} C_VEL
LIN {X 0,Y 573.406,Z 357.081,A -85,B 0,C 180,E1 -2260.06,E2 -2260.06} C_VEL
LIN {X 0,Y 573.52,Z 345.524,A -85,B 0,C 180,E1 -2260.848,E2 -2260.848} C_VEL
LIN {X 0,Y 573.611,Z 333.858,A -85,B 0,C 180,E1 -2261.467,E2 -2261.467} C_VEL
LIN {X 0,Y 573.745,Z 321.147,A -85,B 0,C 180,E1 -2261.975,E2 -2261.975} C_VEL
LIN {X 0,Y 573.864,Z 308.482,A -85,B 0,C 180,E1 -2262.332,E2 -2262.332} C_VEL
LIN {X 0,Y 573.704,Z 303.611,A -85,B 0,C 180,E1 -2262.433,E2 -2262.433} C_VEL
LIN {X 0,Y 573.078,Z 299.527,A -85,B 0,C 180,E1 -2262.529,E2 -2262.529} C_VEL
LIN {X 0,Y 573.156,Z 289.432,A -85,B 0,C 180,E1 -2265.287,E2 -2265.287} C_VEL
LIN {X 0,Y 573.207,Z 278.841,A -85,B 0,C 180,E1 -2268.22,E2 -2268.22} C_VEL
LIN {X 0,Y 573.312,Z 269.574,A -85,B 0,C 180,E1 -2270.825,E2 -2270.825} C_VEL
LIN {X 0,Y 573.375,Z 260.308,A -85,B 0,C 180,E1 -2273.476,E2 -2273.476} C_VEL
LIN {X 0,Y 573.456,Z 251.039,A -85,B 0,C 180,E1 -2276.181,E2 -2276.181} C_VEL
LIN {X 0,Y 573.521,Z 241.772,A -85,B 0,C 180,E1 -2278.95,E2 -2278.95} C_VEL
LIN {X 0,Y 573.697,Z 232.505,A -85,B 0,C 180,E1 -2281.788,E2 -2281.788} C_VEL
LIN {X 0,Y 573.779,Z 224.561,A -85,B 0,C 180,E1 -2284.295,E2 -2284.295} C_VEL
LIN {X 0,Y 573.605,Z 219.232,A -85,B 0,C 180,E1 -2286.035,E2 -2286.035} C_VEL
LIN {X 0,Y 573.237,Z 217.085,A -85,B 0,C 180,E1 -2286.815,E2 -2286.815} C_VEL
LIN {X 0,Y 573.237,Z 217.078,A -85,B 0,C 180,E1 -2289.609,E2 -2289.609} C_VEL
LIN {X 0,Y 573.243,Z 217.079,A -85,B 0,C 180,E1 -2292.642,E2 -2292.642} C_VEL
LIN {X 0,Y 573.243,Z 217.083,A -85,B 0,C 180,E1 -2295.667,E2 -2295.667} C_VEL
LIN {X 0,Y 573.234,Z 217.077,A -85,B 0,C 180,E1 -2298.543,E2 -2298.543} C_VEL
LIN {X 0,Y 573.242,Z 217.082,A -85,B 0,C 180,E1 -2301.298,E2 -2301.298} C_VEL
LIN {X 0,Y 573.19,Z 217.083,A -85,B 0,C 180,E1 -2304.023,E2 -2304.023} C_VEL
LIN {X 0,Y 573.227,Z 217.085,A -85,B 0,C 180,E1 -2306.515,E2 -2306.515} C_VEL
LIN {X 0,Y 573.225,Z 217.078,A -85,B 0,C 180,E1 -2309.12,E2 -2309.12} C_VEL
